(* Usage : 
fbDAIKIN_MasterStation_III_No_1 : FB_BACnet_DAIKIN_MasterStation_III_No_1 :=(Client:=(nDeviceInstance := 1)); 
*)
FUNCTION_BLOCK  FB_BACnet_DAIKIN_MasterStation_III_No_1
VAR_INPUT CONSTANT
	Client : FB_BACnet_Client := (tReadCycleTime:=T#10S,nMaxParallelRequests:=20);
	DAIKIN_MasterStation_III_No_1: FB_BACnetRM_Device := (Client:=Client);
	StartStopCommand_000: FB_BACnetRM_BO := (Client:=Client,nObjectInstance:=1);
	StartStopStatus_000: FB_BACnetRM_BI := (Client:=Client,nObjectInstance:=2);
	Alarm_000: FB_BACnetRM_BI := (Client:=Client,nObjectInstance:=3);
	MalfunctionCode_000: FB_BACnetRM_MI := (Client:=Client,nObjectInstance:=4);
	
	
	
	
	RoomTemp_000: FB_BACnetRM_AI := (Client:=Client,nObjectInstance:=9);
	TempAdjust_000: FB_BACnetRM_AV := (Client:=Client,nObjectInstance:=10);
	FilterSign_000: FB_BACnetRM_BI := (Client:=Client,nObjectInstance:=11);
	FilterSignReset_000: FB_BACnetRM_BV := (Client:=Client,nObjectInstance:=12);
	RemoteControlStart_000: FB_BACnetRM_BV := (Client:=Client,nObjectInstance:=13);
	
	RemoteControlTempAdjust_000: FB_BACnetRM_BV := (Client:=Client,nObjectInstance:=16);
	
	
	
	
	
	
	
	
	
	
	
	
	StartStopCommand_001: FB_BACnetRM_BO := (Client:=Client,nObjectInstance:=257);
	StartStopStatus_001: FB_BACnetRM_BI := (Client:=Client,nObjectInstance:=258);
	Alarm_001: FB_BACnetRM_BI := (Client:=Client,nObjectInstance:=259);
	MalfunctionCode_001: FB_BACnetRM_MI := (Client:=Client,nObjectInstance:=260);
	
	
	
	
	RoomTemp_001: FB_BACnetRM_AI := (Client:=Client,nObjectInstance:=265);
	TempAdjust_001: FB_BACnetRM_AV := (Client:=Client,nObjectInstance:=266);
	FilterSign_001: FB_BACnetRM_BI := (Client:=Client,nObjectInstance:=267);
	FilterSignReset_001: FB_BACnetRM_BV := (Client:=Client,nObjectInstance:=268);
	RemoteControlStart_001: FB_BACnetRM_BV := (Client:=Client,nObjectInstance:=269);
	
	RemoteControlTempAdjust_001: FB_BACnetRM_BV := (Client:=Client,nObjectInstance:=272);
	
	
	
	
	
	
	
	
	
	
	
	
	StartStopCommand_002: FB_BACnetRM_BO := (Client:=Client,nObjectInstance:=513);
	StartStopStatus_002: FB_BACnetRM_BI := (Client:=Client,nObjectInstance:=514);
	Alarm_002: FB_BACnetRM_BI := (Client:=Client,nObjectInstance:=515);
	MalfunctionCode_002: FB_BACnetRM_MI := (Client:=Client,nObjectInstance:=516);
	
	
	
	
	RoomTemp_002: FB_BACnetRM_AI := (Client:=Client,nObjectInstance:=521);
	TempAdjust_002: FB_BACnetRM_AV := (Client:=Client,nObjectInstance:=522);
	FilterSign_002: FB_BACnetRM_BI := (Client:=Client,nObjectInstance:=523);
	FilterSignReset_002: FB_BACnetRM_BV := (Client:=Client,nObjectInstance:=524);
	RemoteControlStart_002: FB_BACnetRM_BV := (Client:=Client,nObjectInstance:=525);
	
	RemoteControlTempAdjust_002: FB_BACnetRM_BV := (Client:=Client,nObjectInstance:=528);
	
	
	
	
	
	
	
	
	
	
	
	
	StartStopCommand_003: FB_BACnetRM_BO := (Client:=Client,nObjectInstance:=769);
	StartStopStatus_003: FB_BACnetRM_BI := (Client:=Client,nObjectInstance:=770);
	Alarm_003: FB_BACnetRM_BI := (Client:=Client,nObjectInstance:=771);
	MalfunctionCode_003: FB_BACnetRM_MI := (Client:=Client,nObjectInstance:=772);
	
	
	
	
	RoomTemp_003: FB_BACnetRM_AI := (Client:=Client,nObjectInstance:=777);
	TempAdjust_003: FB_BACnetRM_AV := (Client:=Client,nObjectInstance:=778);
	FilterSign_003: FB_BACnetRM_BI := (Client:=Client,nObjectInstance:=779);
	FilterSignReset_003: FB_BACnetRM_BV := (Client:=Client,nObjectInstance:=780);
	RemoteControlStart_003: FB_BACnetRM_BV := (Client:=Client,nObjectInstance:=781);
	
	RemoteControlTempAdjust_003: FB_BACnetRM_BV := (Client:=Client,nObjectInstance:=784);
	
	
	
	
	
	
	
	
	
	
	
	
	StartStopCommand_004: FB_BACnetRM_BO := (Client:=Client,nObjectInstance:=1025);
	StartStopStatus_004: FB_BACnetRM_BI := (Client:=Client,nObjectInstance:=1026);
	Alarm_004: FB_BACnetRM_BI := (Client:=Client,nObjectInstance:=1027);
	MalfunctionCode_004: FB_BACnetRM_MI := (Client:=Client,nObjectInstance:=1028);
	
	
	
	
	RoomTemp_004: FB_BACnetRM_AI := (Client:=Client,nObjectInstance:=1033);
	TempAdjust_004: FB_BACnetRM_AV := (Client:=Client,nObjectInstance:=1034);
	FilterSign_004: FB_BACnetRM_BI := (Client:=Client,nObjectInstance:=1035);
	FilterSignReset_004: FB_BACnetRM_BV := (Client:=Client,nObjectInstance:=1036);
	RemoteControlStart_004: FB_BACnetRM_BV := (Client:=Client,nObjectInstance:=1037);
	
	RemoteControlTempAdjust_004: FB_BACnetRM_BV := (Client:=Client,nObjectInstance:=1040);
	
	
	
	
	
	
	
	
	
	
	
	
	StartStopCommand_005: FB_BACnetRM_BO := (Client:=Client,nObjectInstance:=1281);
	StartStopStatus_005: FB_BACnetRM_BI := (Client:=Client,nObjectInstance:=1282);
	Alarm_005: FB_BACnetRM_BI := (Client:=Client,nObjectInstance:=1283);
	MalfunctionCode_005: FB_BACnetRM_MI := (Client:=Client,nObjectInstance:=1284);
	
	
	
	
	RoomTemp_005: FB_BACnetRM_AI := (Client:=Client,nObjectInstance:=1289);
	TempAdjust_005: FB_BACnetRM_AV := (Client:=Client,nObjectInstance:=1290);
	FilterSign_005: FB_BACnetRM_BI := (Client:=Client,nObjectInstance:=1291);
	FilterSignReset_005: FB_BACnetRM_BV := (Client:=Client,nObjectInstance:=1292);
	RemoteControlStart_005: FB_BACnetRM_BV := (Client:=Client,nObjectInstance:=1293);
	
	RemoteControlTempAdjust_005: FB_BACnetRM_BV := (Client:=Client,nObjectInstance:=1296);
	
	
	
	
	
	
	
	
	
	
	
	
	StartStopCommand_006: FB_BACnetRM_BO := (Client:=Client,nObjectInstance:=1537);
	StartStopStatus_006: FB_BACnetRM_BI := (Client:=Client,nObjectInstance:=1538);
	Alarm_006: FB_BACnetRM_BI := (Client:=Client,nObjectInstance:=1539);
	MalfunctionCode_006: FB_BACnetRM_MI := (Client:=Client,nObjectInstance:=1540);
	
	
	
	
	RoomTemp_006: FB_BACnetRM_AI := (Client:=Client,nObjectInstance:=1545);
	TempAdjust_006: FB_BACnetRM_AV := (Client:=Client,nObjectInstance:=1546);
	FilterSign_006: FB_BACnetRM_BI := (Client:=Client,nObjectInstance:=1547);
	FilterSignReset_006: FB_BACnetRM_BV := (Client:=Client,nObjectInstance:=1548);
	RemoteControlStart_006: FB_BACnetRM_BV := (Client:=Client,nObjectInstance:=1549);
	
	RemoteControlTempAdjust_006: FB_BACnetRM_BV := (Client:=Client,nObjectInstance:=1552);
	
	
	
	
	
	
	
	
	
	
	
	
	StartStopCommand_007: FB_BACnetRM_BO := (Client:=Client,nObjectInstance:=1793);
	StartStopStatus_007: FB_BACnetRM_BI := (Client:=Client,nObjectInstance:=1794);
	Alarm_007: FB_BACnetRM_BI := (Client:=Client,nObjectInstance:=1795);
	MalfunctionCode_007: FB_BACnetRM_MI := (Client:=Client,nObjectInstance:=1796);
	
	
	
	
	RoomTemp_007: FB_BACnetRM_AI := (Client:=Client,nObjectInstance:=1801);
	TempAdjust_007: FB_BACnetRM_AV := (Client:=Client,nObjectInstance:=1802);
	FilterSign_007: FB_BACnetRM_BI := (Client:=Client,nObjectInstance:=1803);
	FilterSignReset_007: FB_BACnetRM_BV := (Client:=Client,nObjectInstance:=1804);
	RemoteControlStart_007: FB_BACnetRM_BV := (Client:=Client,nObjectInstance:=1805);
	
	RemoteControlTempAdjust_007: FB_BACnetRM_BV := (Client:=Client,nObjectInstance:=1808);
	
	
	
	
	
	
	
	
	
	
	
	
	StartStopCommand_008: FB_BACnetRM_BO := (Client:=Client,nObjectInstance:=2049);
	StartStopStatus_008: FB_BACnetRM_BI := (Client:=Client,nObjectInstance:=2050);
	Alarm_008: FB_BACnetRM_BI := (Client:=Client,nObjectInstance:=2051);
	MalfunctionCode_008: FB_BACnetRM_MI := (Client:=Client,nObjectInstance:=2052);
	
	
	
	
	RoomTemp_008: FB_BACnetRM_AI := (Client:=Client,nObjectInstance:=2057);
	TempAdjust_008: FB_BACnetRM_AV := (Client:=Client,nObjectInstance:=2058);
	FilterSign_008: FB_BACnetRM_BI := (Client:=Client,nObjectInstance:=2059);
	FilterSignReset_008: FB_BACnetRM_BV := (Client:=Client,nObjectInstance:=2060);
	RemoteControlStart_008: FB_BACnetRM_BV := (Client:=Client,nObjectInstance:=2061);
	
	RemoteControlTempAdjust_008: FB_BACnetRM_BV := (Client:=Client,nObjectInstance:=2064);
	
	
	
	
	
	
	
	
	
	
	
	
	StartStopCommand_009: FB_BACnetRM_BO := (Client:=Client,nObjectInstance:=2305);
	StartStopStatus_009: FB_BACnetRM_BI := (Client:=Client,nObjectInstance:=2306);
	Alarm_009: FB_BACnetRM_BI := (Client:=Client,nObjectInstance:=2307);
	MalfunctionCode_009: FB_BACnetRM_MI := (Client:=Client,nObjectInstance:=2308);
	
	
	
	
	RoomTemp_009: FB_BACnetRM_AI := (Client:=Client,nObjectInstance:=2313);
	TempAdjust_009: FB_BACnetRM_AV := (Client:=Client,nObjectInstance:=2314);
	FilterSign_009: FB_BACnetRM_BI := (Client:=Client,nObjectInstance:=2315);
	FilterSignReset_009: FB_BACnetRM_BV := (Client:=Client,nObjectInstance:=2316);
	RemoteControlStart_009: FB_BACnetRM_BV := (Client:=Client,nObjectInstance:=2317);
	
	RemoteControlTempAdjust_009: FB_BACnetRM_BV := (Client:=Client,nObjectInstance:=2320);
	
	
	
	
	
	
	
	
	
	
	
	
	StartStopCommand_010: FB_BACnetRM_BO := (Client:=Client,nObjectInstance:=2561);
	StartStopStatus_010: FB_BACnetRM_BI := (Client:=Client,nObjectInstance:=2562);
	Alarm_010: FB_BACnetRM_BI := (Client:=Client,nObjectInstance:=2563);
	MalfunctionCode_010: FB_BACnetRM_MI := (Client:=Client,nObjectInstance:=2564);
	
	
	
	
	RoomTemp_010: FB_BACnetRM_AI := (Client:=Client,nObjectInstance:=2569);
	TempAdjust_010: FB_BACnetRM_AV := (Client:=Client,nObjectInstance:=2570);
	FilterSign_010: FB_BACnetRM_BI := (Client:=Client,nObjectInstance:=2571);
	FilterSignReset_010: FB_BACnetRM_BV := (Client:=Client,nObjectInstance:=2572);
	RemoteControlStart_010: FB_BACnetRM_BV := (Client:=Client,nObjectInstance:=2573);
	
	RemoteControlTempAdjust_010: FB_BACnetRM_BV := (Client:=Client,nObjectInstance:=2576);
	
	
	
	
	
	
	
	
	
	
	
	
	StartStopCommand_011: FB_BACnetRM_BO := (Client:=Client,nObjectInstance:=2817);
	StartStopStatus_011: FB_BACnetRM_BI := (Client:=Client,nObjectInstance:=2818);
	Alarm_011: FB_BACnetRM_BI := (Client:=Client,nObjectInstance:=2819);
	MalfunctionCode_011: FB_BACnetRM_MI := (Client:=Client,nObjectInstance:=2820);
	
	
	
	
	RoomTemp_011: FB_BACnetRM_AI := (Client:=Client,nObjectInstance:=2825);
	TempAdjust_011: FB_BACnetRM_AV := (Client:=Client,nObjectInstance:=2826);
	FilterSign_011: FB_BACnetRM_BI := (Client:=Client,nObjectInstance:=2827);
	FilterSignReset_011: FB_BACnetRM_BV := (Client:=Client,nObjectInstance:=2828);
	RemoteControlStart_011: FB_BACnetRM_BV := (Client:=Client,nObjectInstance:=2829);
	
	RemoteControlTempAdjust_011: FB_BACnetRM_BV := (Client:=Client,nObjectInstance:=2832);
	
	
	
	
	
	
	
	
	
	
	
	
	StartStopCommand_012: FB_BACnetRM_BO := (Client:=Client,nObjectInstance:=3073);
	StartStopStatus_012: FB_BACnetRM_BI := (Client:=Client,nObjectInstance:=3074);
	Alarm_012: FB_BACnetRM_BI := (Client:=Client,nObjectInstance:=3075);
	MalfunctionCode_012: FB_BACnetRM_MI := (Client:=Client,nObjectInstance:=3076);
	
	
	
	
	RoomTemp_012: FB_BACnetRM_AI := (Client:=Client,nObjectInstance:=3081);
	TempAdjust_012: FB_BACnetRM_AV := (Client:=Client,nObjectInstance:=3082);
	FilterSign_012: FB_BACnetRM_BI := (Client:=Client,nObjectInstance:=3083);
	FilterSignReset_012: FB_BACnetRM_BV := (Client:=Client,nObjectInstance:=3084);
	RemoteControlStart_012: FB_BACnetRM_BV := (Client:=Client,nObjectInstance:=3085);
	
	RemoteControlTempAdjust_012: FB_BACnetRM_BV := (Client:=Client,nObjectInstance:=3088);
	
	
	
	
	
	
	
	
	
	
	
	
	StartStopCommand_013: FB_BACnetRM_BO := (Client:=Client,nObjectInstance:=3329);
	StartStopStatus_013: FB_BACnetRM_BI := (Client:=Client,nObjectInstance:=3330);
	Alarm_013: FB_BACnetRM_BI := (Client:=Client,nObjectInstance:=3331);
	MalfunctionCode_013: FB_BACnetRM_MI := (Client:=Client,nObjectInstance:=3332);
	
	
	
	
	RoomTemp_013: FB_BACnetRM_AI := (Client:=Client,nObjectInstance:=3337);
	TempAdjust_013: FB_BACnetRM_AV := (Client:=Client,nObjectInstance:=3338);
	FilterSign_013: FB_BACnetRM_BI := (Client:=Client,nObjectInstance:=3339);
	FilterSignReset_013: FB_BACnetRM_BV := (Client:=Client,nObjectInstance:=3340);
	RemoteControlStart_013: FB_BACnetRM_BV := (Client:=Client,nObjectInstance:=3341);
	
	RemoteControlTempAdjust_013: FB_BACnetRM_BV := (Client:=Client,nObjectInstance:=3344);
	
	
	
	
	
	
	
	
	
	
	
	
	StartStopCommand_014: FB_BACnetRM_BO := (Client:=Client,nObjectInstance:=3585);
	StartStopStatus_014: FB_BACnetRM_BI := (Client:=Client,nObjectInstance:=3586);
	Alarm_014: FB_BACnetRM_BI := (Client:=Client,nObjectInstance:=3587);
	MalfunctionCode_014: FB_BACnetRM_MI := (Client:=Client,nObjectInstance:=3588);
	
	
	
	
	RoomTemp_014: FB_BACnetRM_AI := (Client:=Client,nObjectInstance:=3593);
	TempAdjust_014: FB_BACnetRM_AV := (Client:=Client,nObjectInstance:=3594);
	FilterSign_014: FB_BACnetRM_BI := (Client:=Client,nObjectInstance:=3595);
	FilterSignReset_014: FB_BACnetRM_BV := (Client:=Client,nObjectInstance:=3596);
	RemoteControlStart_014: FB_BACnetRM_BV := (Client:=Client,nObjectInstance:=3597);
	
	RemoteControlTempAdjust_014: FB_BACnetRM_BV := (Client:=Client,nObjectInstance:=3600);
	
	
	
	
	
	
	
	
	
	
	
	
	StartStopCommand_015: FB_BACnetRM_BO := (Client:=Client,nObjectInstance:=3841);
	StartStopStatus_015: FB_BACnetRM_BI := (Client:=Client,nObjectInstance:=3842);
	Alarm_015: FB_BACnetRM_BI := (Client:=Client,nObjectInstance:=3843);
	MalfunctionCode_015: FB_BACnetRM_MI := (Client:=Client,nObjectInstance:=3844);
	
	
	
	
	RoomTemp_015: FB_BACnetRM_AI := (Client:=Client,nObjectInstance:=3849);
	TempAdjust_015: FB_BACnetRM_AV := (Client:=Client,nObjectInstance:=3850);
	FilterSign_015: FB_BACnetRM_BI := (Client:=Client,nObjectInstance:=3851);
	FilterSignReset_015: FB_BACnetRM_BV := (Client:=Client,nObjectInstance:=3852);
	RemoteControlStart_015: FB_BACnetRM_BV := (Client:=Client,nObjectInstance:=3853);
	
	RemoteControlTempAdjust_015: FB_BACnetRM_BV := (Client:=Client,nObjectInstance:=3856);
	
	
	
	
	
	
	
	
	
	
	
	
	StartStopCommand_016: FB_BACnetRM_BO := (Client:=Client,nObjectInstance:=4097);
	StartStopStatus_016: FB_BACnetRM_BI := (Client:=Client,nObjectInstance:=4098);
	Alarm_016: FB_BACnetRM_BI := (Client:=Client,nObjectInstance:=4099);
	MalfunctionCode_016: FB_BACnetRM_MI := (Client:=Client,nObjectInstance:=4100);
	
	
	
	
	RoomTemp_016: FB_BACnetRM_AI := (Client:=Client,nObjectInstance:=4105);
	TempAdjust_016: FB_BACnetRM_AV := (Client:=Client,nObjectInstance:=4106);
	FilterSign_016: FB_BACnetRM_BI := (Client:=Client,nObjectInstance:=4107);
	FilterSignReset_016: FB_BACnetRM_BV := (Client:=Client,nObjectInstance:=4108);
	RemoteControlStart_016: FB_BACnetRM_BV := (Client:=Client,nObjectInstance:=4109);
	
	RemoteControlTempAdjust_016: FB_BACnetRM_BV := (Client:=Client,nObjectInstance:=4112);
	
	
	
	
	
	
	
	
	
	
	
	
	StartStopCommand_017: FB_BACnetRM_BO := (Client:=Client,nObjectInstance:=4353);
	StartStopStatus_017: FB_BACnetRM_BI := (Client:=Client,nObjectInstance:=4354);
	Alarm_017: FB_BACnetRM_BI := (Client:=Client,nObjectInstance:=4355);
	MalfunctionCode_017: FB_BACnetRM_MI := (Client:=Client,nObjectInstance:=4356);
	
	
	
	
	RoomTemp_017: FB_BACnetRM_AI := (Client:=Client,nObjectInstance:=4361);
	TempAdjust_017: FB_BACnetRM_AV := (Client:=Client,nObjectInstance:=4362);
	FilterSign_017: FB_BACnetRM_BI := (Client:=Client,nObjectInstance:=4363);
	FilterSignReset_017: FB_BACnetRM_BV := (Client:=Client,nObjectInstance:=4364);
	RemoteControlStart_017: FB_BACnetRM_BV := (Client:=Client,nObjectInstance:=4365);
	
	RemoteControlTempAdjust_017: FB_BACnetRM_BV := (Client:=Client,nObjectInstance:=4368);
	
	
	
	
	
	
	
	
	
	
	
	
	StartStopCommand_018: FB_BACnetRM_BO := (Client:=Client,nObjectInstance:=4609);
	StartStopStatus_018: FB_BACnetRM_BI := (Client:=Client,nObjectInstance:=4610);
	Alarm_018: FB_BACnetRM_BI := (Client:=Client,nObjectInstance:=4611);
	MalfunctionCode_018: FB_BACnetRM_MI := (Client:=Client,nObjectInstance:=4612);
	
	
	
	
	RoomTemp_018: FB_BACnetRM_AI := (Client:=Client,nObjectInstance:=4617);
	TempAdjust_018: FB_BACnetRM_AV := (Client:=Client,nObjectInstance:=4618);
	FilterSign_018: FB_BACnetRM_BI := (Client:=Client,nObjectInstance:=4619);
	FilterSignReset_018: FB_BACnetRM_BV := (Client:=Client,nObjectInstance:=4620);
	RemoteControlStart_018: FB_BACnetRM_BV := (Client:=Client,nObjectInstance:=4621);
	
	RemoteControlTempAdjust_018: FB_BACnetRM_BV := (Client:=Client,nObjectInstance:=4624);
	
	
	
	
	
	
	
	
	
	
	
	
	StartStopCommand_019: FB_BACnetRM_BO := (Client:=Client,nObjectInstance:=4865);
	StartStopStatus_019: FB_BACnetRM_BI := (Client:=Client,nObjectInstance:=4866);
	Alarm_019: FB_BACnetRM_BI := (Client:=Client,nObjectInstance:=4867);
	MalfunctionCode_019: FB_BACnetRM_MI := (Client:=Client,nObjectInstance:=4868);
	
	
	
	
	RoomTemp_019: FB_BACnetRM_AI := (Client:=Client,nObjectInstance:=4873);
	TempAdjust_019: FB_BACnetRM_AV := (Client:=Client,nObjectInstance:=4874);
	FilterSign_019: FB_BACnetRM_BI := (Client:=Client,nObjectInstance:=4875);
	FilterSignReset_019: FB_BACnetRM_BV := (Client:=Client,nObjectInstance:=4876);
	RemoteControlStart_019: FB_BACnetRM_BV := (Client:=Client,nObjectInstance:=4877);
	
	RemoteControlTempAdjust_019: FB_BACnetRM_BV := (Client:=Client,nObjectInstance:=4880);
	
	
	
	
	
	
	
	
	
	
	
	
	StartStopCommand_020: FB_BACnetRM_BO := (Client:=Client,nObjectInstance:=5121);
	StartStopStatus_020: FB_BACnetRM_BI := (Client:=Client,nObjectInstance:=5122);
	Alarm_020: FB_BACnetRM_BI := (Client:=Client,nObjectInstance:=5123);
	MalfunctionCode_020: FB_BACnetRM_MI := (Client:=Client,nObjectInstance:=5124);
	
	
	
	
	RoomTemp_020: FB_BACnetRM_AI := (Client:=Client,nObjectInstance:=5129);
	TempAdjust_020: FB_BACnetRM_AV := (Client:=Client,nObjectInstance:=5130);
	FilterSign_020: FB_BACnetRM_BI := (Client:=Client,nObjectInstance:=5131);
	FilterSignReset_020: FB_BACnetRM_BV := (Client:=Client,nObjectInstance:=5132);
	RemoteControlStart_020: FB_BACnetRM_BV := (Client:=Client,nObjectInstance:=5133);
	
	RemoteControlTempAdjust_020: FB_BACnetRM_BV := (Client:=Client,nObjectInstance:=5136);
	
	
	
	
	
	
	
	
	
	
	
	
	StartStopCommand_021: FB_BACnetRM_BO := (Client:=Client,nObjectInstance:=5377);
	StartStopStatus_021: FB_BACnetRM_BI := (Client:=Client,nObjectInstance:=5378);
	Alarm_021: FB_BACnetRM_BI := (Client:=Client,nObjectInstance:=5379);
	MalfunctionCode_021: FB_BACnetRM_MI := (Client:=Client,nObjectInstance:=5380);
	
	
	
	
	RoomTemp_021: FB_BACnetRM_AI := (Client:=Client,nObjectInstance:=5385);
	TempAdjust_021: FB_BACnetRM_AV := (Client:=Client,nObjectInstance:=5386);
	FilterSign_021: FB_BACnetRM_BI := (Client:=Client,nObjectInstance:=5387);
	FilterSignReset_021: FB_BACnetRM_BV := (Client:=Client,nObjectInstance:=5388);
	RemoteControlStart_021: FB_BACnetRM_BV := (Client:=Client,nObjectInstance:=5389);
	
	RemoteControlTempAdjust_021: FB_BACnetRM_BV := (Client:=Client,nObjectInstance:=5392);
	
	
	
	
	
	
	
	
	
	
	
	
	StartStopCommand_022: FB_BACnetRM_BO := (Client:=Client,nObjectInstance:=5633);
	StartStopStatus_022: FB_BACnetRM_BI := (Client:=Client,nObjectInstance:=5634);
	Alarm_022: FB_BACnetRM_BI := (Client:=Client,nObjectInstance:=5635);
	MalfunctionCode_022: FB_BACnetRM_MI := (Client:=Client,nObjectInstance:=5636);
	
	
	
	
	RoomTemp_022: FB_BACnetRM_AI := (Client:=Client,nObjectInstance:=5641);
	TempAdjust_022: FB_BACnetRM_AV := (Client:=Client,nObjectInstance:=5642);
	FilterSign_022: FB_BACnetRM_BI := (Client:=Client,nObjectInstance:=5643);
	FilterSignReset_022: FB_BACnetRM_BV := (Client:=Client,nObjectInstance:=5644);
	RemoteControlStart_022: FB_BACnetRM_BV := (Client:=Client,nObjectInstance:=5645);
	
	RemoteControlTempAdjust_022: FB_BACnetRM_BV := (Client:=Client,nObjectInstance:=5648);
	
	
	
	
	
	
	
	
	
	
	
	
	StartStopCommand_023: FB_BACnetRM_BO := (Client:=Client,nObjectInstance:=5889);
	StartStopStatus_023: FB_BACnetRM_BI := (Client:=Client,nObjectInstance:=5890);
	Alarm_023: FB_BACnetRM_BI := (Client:=Client,nObjectInstance:=5891);
	MalfunctionCode_023: FB_BACnetRM_MI := (Client:=Client,nObjectInstance:=5892);
	
	
	
	
	RoomTemp_023: FB_BACnetRM_AI := (Client:=Client,nObjectInstance:=5897);
	TempAdjust_023: FB_BACnetRM_AV := (Client:=Client,nObjectInstance:=5898);
	FilterSign_023: FB_BACnetRM_BI := (Client:=Client,nObjectInstance:=5899);
	FilterSignReset_023: FB_BACnetRM_BV := (Client:=Client,nObjectInstance:=5900);
	RemoteControlStart_023: FB_BACnetRM_BV := (Client:=Client,nObjectInstance:=5901);
	
	RemoteControlTempAdjust_023: FB_BACnetRM_BV := (Client:=Client,nObjectInstance:=5904);
	
	
	
	
	
	
	
	
	
	
	
	
	StartStopCommand_024: FB_BACnetRM_BO := (Client:=Client,nObjectInstance:=6145);
	StartStopStatus_024: FB_BACnetRM_BI := (Client:=Client,nObjectInstance:=6146);
	Alarm_024: FB_BACnetRM_BI := (Client:=Client,nObjectInstance:=6147);
	MalfunctionCode_024: FB_BACnetRM_MI := (Client:=Client,nObjectInstance:=6148);
	
	
	
	
	RoomTemp_024: FB_BACnetRM_AI := (Client:=Client,nObjectInstance:=6153);
	TempAdjust_024: FB_BACnetRM_AV := (Client:=Client,nObjectInstance:=6154);
	FilterSign_024: FB_BACnetRM_BI := (Client:=Client,nObjectInstance:=6155);
	FilterSignReset_024: FB_BACnetRM_BV := (Client:=Client,nObjectInstance:=6156);
	RemoteControlStart_024: FB_BACnetRM_BV := (Client:=Client,nObjectInstance:=6157);
	
	RemoteControlTempAdjust_024: FB_BACnetRM_BV := (Client:=Client,nObjectInstance:=6160);
	
	
	
	
	
	
	
	
	
	
	
	
	StartStopCommand_025: FB_BACnetRM_BO := (Client:=Client,nObjectInstance:=6401);
	StartStopStatus_025: FB_BACnetRM_BI := (Client:=Client,nObjectInstance:=6402);
	Alarm_025: FB_BACnetRM_BI := (Client:=Client,nObjectInstance:=6403);
	MalfunctionCode_025: FB_BACnetRM_MI := (Client:=Client,nObjectInstance:=6404);
	
	
	
	
	RoomTemp_025: FB_BACnetRM_AI := (Client:=Client,nObjectInstance:=6409);
	TempAdjust_025: FB_BACnetRM_AV := (Client:=Client,nObjectInstance:=6410);
	FilterSign_025: FB_BACnetRM_BI := (Client:=Client,nObjectInstance:=6411);
	FilterSignReset_025: FB_BACnetRM_BV := (Client:=Client,nObjectInstance:=6412);
	RemoteControlStart_025: FB_BACnetRM_BV := (Client:=Client,nObjectInstance:=6413);
	
	RemoteControlTempAdjust_025: FB_BACnetRM_BV := (Client:=Client,nObjectInstance:=6416);
	
	
	
	
	
	
	
	
	
	
	
	
	StartStopCommand_026: FB_BACnetRM_BO := (Client:=Client,nObjectInstance:=6657);
	StartStopStatus_026: FB_BACnetRM_BI := (Client:=Client,nObjectInstance:=6658);
	Alarm_026: FB_BACnetRM_BI := (Client:=Client,nObjectInstance:=6659);
	MalfunctionCode_026: FB_BACnetRM_MI := (Client:=Client,nObjectInstance:=6660);
	
	
	
	
	RoomTemp_026: FB_BACnetRM_AI := (Client:=Client,nObjectInstance:=6665);
	TempAdjust_026: FB_BACnetRM_AV := (Client:=Client,nObjectInstance:=6666);
	FilterSign_026: FB_BACnetRM_BI := (Client:=Client,nObjectInstance:=6667);
	FilterSignReset_026: FB_BACnetRM_BV := (Client:=Client,nObjectInstance:=6668);
	RemoteControlStart_026: FB_BACnetRM_BV := (Client:=Client,nObjectInstance:=6669);
	
	RemoteControlTempAdjust_026: FB_BACnetRM_BV := (Client:=Client,nObjectInstance:=6672);
	
	
	
	
	
	
	
	
	
	
	
	
	StartStopCommand_027: FB_BACnetRM_BO := (Client:=Client,nObjectInstance:=6913);
	StartStopStatus_027: FB_BACnetRM_BI := (Client:=Client,nObjectInstance:=6914);
	Alarm_027: FB_BACnetRM_BI := (Client:=Client,nObjectInstance:=6915);
	MalfunctionCode_027: FB_BACnetRM_MI := (Client:=Client,nObjectInstance:=6916);
	
	
	
	
	RoomTemp_027: FB_BACnetRM_AI := (Client:=Client,nObjectInstance:=6921);
	TempAdjust_027: FB_BACnetRM_AV := (Client:=Client,nObjectInstance:=6922);
	FilterSign_027: FB_BACnetRM_BI := (Client:=Client,nObjectInstance:=6923);
	FilterSignReset_027: FB_BACnetRM_BV := (Client:=Client,nObjectInstance:=6924);
	RemoteControlStart_027: FB_BACnetRM_BV := (Client:=Client,nObjectInstance:=6925);
	
	RemoteControlTempAdjust_027: FB_BACnetRM_BV := (Client:=Client,nObjectInstance:=6928);
	
	
	
	
	
	
	
	
	
	
	
	
	StartStopCommand_028: FB_BACnetRM_BO := (Client:=Client,nObjectInstance:=7169);
	StartStopStatus_028: FB_BACnetRM_BI := (Client:=Client,nObjectInstance:=7170);
	Alarm_028: FB_BACnetRM_BI := (Client:=Client,nObjectInstance:=7171);
	MalfunctionCode_028: FB_BACnetRM_MI := (Client:=Client,nObjectInstance:=7172);
	
	
	
	
	RoomTemp_028: FB_BACnetRM_AI := (Client:=Client,nObjectInstance:=7177);
	TempAdjust_028: FB_BACnetRM_AV := (Client:=Client,nObjectInstance:=7178);
	FilterSign_028: FB_BACnetRM_BI := (Client:=Client,nObjectInstance:=7179);
	FilterSignReset_028: FB_BACnetRM_BV := (Client:=Client,nObjectInstance:=7180);
	RemoteControlStart_028: FB_BACnetRM_BV := (Client:=Client,nObjectInstance:=7181);
	
	RemoteControlTempAdjust_028: FB_BACnetRM_BV := (Client:=Client,nObjectInstance:=7184);
	
	
	
	
	
	
	
	
	
	
	
	
	StartStopCommand_029: FB_BACnetRM_BO := (Client:=Client,nObjectInstance:=7425);
	StartStopStatus_029: FB_BACnetRM_BI := (Client:=Client,nObjectInstance:=7426);
	Alarm_029: FB_BACnetRM_BI := (Client:=Client,nObjectInstance:=7427);
	MalfunctionCode_029: FB_BACnetRM_MI := (Client:=Client,nObjectInstance:=7428);
	
	
	
	
	RoomTemp_029: FB_BACnetRM_AI := (Client:=Client,nObjectInstance:=7433);
	TempAdjust_029: FB_BACnetRM_AV := (Client:=Client,nObjectInstance:=7434);
	FilterSign_029: FB_BACnetRM_BI := (Client:=Client,nObjectInstance:=7435);
	FilterSignReset_029: FB_BACnetRM_BV := (Client:=Client,nObjectInstance:=7436);
	RemoteControlStart_029: FB_BACnetRM_BV := (Client:=Client,nObjectInstance:=7437);
	
	RemoteControlTempAdjust_029: FB_BACnetRM_BV := (Client:=Client,nObjectInstance:=7440);
	
	
	
	
	
	
	
	
	
	
	
	
	StartStopCommand_030: FB_BACnetRM_BO := (Client:=Client,nObjectInstance:=7681);
	StartStopStatus_030: FB_BACnetRM_BI := (Client:=Client,nObjectInstance:=7682);
	Alarm_030: FB_BACnetRM_BI := (Client:=Client,nObjectInstance:=7683);
	MalfunctionCode_030: FB_BACnetRM_MI := (Client:=Client,nObjectInstance:=7684);
	
	
	
	
	RoomTemp_030: FB_BACnetRM_AI := (Client:=Client,nObjectInstance:=7689);
	TempAdjust_030: FB_BACnetRM_AV := (Client:=Client,nObjectInstance:=7690);
	FilterSign_030: FB_BACnetRM_BI := (Client:=Client,nObjectInstance:=7691);
	FilterSignReset_030: FB_BACnetRM_BV := (Client:=Client,nObjectInstance:=7692);
	RemoteControlStart_030: FB_BACnetRM_BV := (Client:=Client,nObjectInstance:=7693);
	
	RemoteControlTempAdjust_030: FB_BACnetRM_BV := (Client:=Client,nObjectInstance:=7696);
	
	
	
	
	
	
	
	
	
	
	
	
	StartStopCommand_031: FB_BACnetRM_BO := (Client:=Client,nObjectInstance:=7937);
	StartStopStatus_031: FB_BACnetRM_BI := (Client:=Client,nObjectInstance:=7938);
	Alarm_031: FB_BACnetRM_BI := (Client:=Client,nObjectInstance:=7939);
	MalfunctionCode_031: FB_BACnetRM_MI := (Client:=Client,nObjectInstance:=7940);
	
	
	
	
	RoomTemp_031: FB_BACnetRM_AI := (Client:=Client,nObjectInstance:=7945);
	TempAdjust_031: FB_BACnetRM_AV := (Client:=Client,nObjectInstance:=7946);
	FilterSign_031: FB_BACnetRM_BI := (Client:=Client,nObjectInstance:=7947);
	FilterSignReset_031: FB_BACnetRM_BV := (Client:=Client,nObjectInstance:=7948);
	RemoteControlStart_031: FB_BACnetRM_BV := (Client:=Client,nObjectInstance:=7949);
	
	RemoteControlTempAdjust_031: FB_BACnetRM_BV := (Client:=Client,nObjectInstance:=7952);
	
	
	
	
	
	
	
	
	
	
	
	
	StartStopCommand_032: FB_BACnetRM_BO := (Client:=Client,nObjectInstance:=8193);
	StartStopStatus_032: FB_BACnetRM_BI := (Client:=Client,nObjectInstance:=8194);
	Alarm_032: FB_BACnetRM_BI := (Client:=Client,nObjectInstance:=8195);
	MalfunctionCode_032: FB_BACnetRM_MI := (Client:=Client,nObjectInstance:=8196);
	
	
	
	
	RoomTemp_032: FB_BACnetRM_AI := (Client:=Client,nObjectInstance:=8201);
	TempAdjust_032: FB_BACnetRM_AV := (Client:=Client,nObjectInstance:=8202);
	FilterSign_032: FB_BACnetRM_BI := (Client:=Client,nObjectInstance:=8203);
	FilterSignReset_032: FB_BACnetRM_BV := (Client:=Client,nObjectInstance:=8204);
	RemoteControlStart_032: FB_BACnetRM_BV := (Client:=Client,nObjectInstance:=8205);
	
	RemoteControlTempAdjust_032: FB_BACnetRM_BV := (Client:=Client,nObjectInstance:=8208);
	
	
	
	
	
	
	
	
	
	
	
	
	StartStopCommand_033: FB_BACnetRM_BO := (Client:=Client,nObjectInstance:=8449);
	StartStopStatus_033: FB_BACnetRM_BI := (Client:=Client,nObjectInstance:=8450);
	Alarm_033: FB_BACnetRM_BI := (Client:=Client,nObjectInstance:=8451);
	MalfunctionCode_033: FB_BACnetRM_MI := (Client:=Client,nObjectInstance:=8452);
	
	
	
	
	RoomTemp_033: FB_BACnetRM_AI := (Client:=Client,nObjectInstance:=8457);
	TempAdjust_033: FB_BACnetRM_AV := (Client:=Client,nObjectInstance:=8458);
	FilterSign_033: FB_BACnetRM_BI := (Client:=Client,nObjectInstance:=8459);
	FilterSignReset_033: FB_BACnetRM_BV := (Client:=Client,nObjectInstance:=8460);
	RemoteControlStart_033: FB_BACnetRM_BV := (Client:=Client,nObjectInstance:=8461);
	
	RemoteControlTempAdjust_033: FB_BACnetRM_BV := (Client:=Client,nObjectInstance:=8464);
	
	
	
	
	
	
	
	
	
	
	
	
	StartStopCommand_034: FB_BACnetRM_BO := (Client:=Client,nObjectInstance:=8705);
	StartStopStatus_034: FB_BACnetRM_BI := (Client:=Client,nObjectInstance:=8706);
	Alarm_034: FB_BACnetRM_BI := (Client:=Client,nObjectInstance:=8707);
	MalfunctionCode_034: FB_BACnetRM_MI := (Client:=Client,nObjectInstance:=8708);
	
	
	
	
	RoomTemp_034: FB_BACnetRM_AI := (Client:=Client,nObjectInstance:=8713);
	TempAdjust_034: FB_BACnetRM_AV := (Client:=Client,nObjectInstance:=8714);
	FilterSign_034: FB_BACnetRM_BI := (Client:=Client,nObjectInstance:=8715);
	FilterSignReset_034: FB_BACnetRM_BV := (Client:=Client,nObjectInstance:=8716);
	RemoteControlStart_034: FB_BACnetRM_BV := (Client:=Client,nObjectInstance:=8717);
	
	RemoteControlTempAdjust_034: FB_BACnetRM_BV := (Client:=Client,nObjectInstance:=8720);
	
	
	
	
	
	
	
	
	
	
	
	
	StartStopCommand_035: FB_BACnetRM_BO := (Client:=Client,nObjectInstance:=8961);
	StartStopStatus_035: FB_BACnetRM_BI := (Client:=Client,nObjectInstance:=8962);
	Alarm_035: FB_BACnetRM_BI := (Client:=Client,nObjectInstance:=8963);
	MalfunctionCode_035: FB_BACnetRM_MI := (Client:=Client,nObjectInstance:=8964);
	
	
	
	
	RoomTemp_035: FB_BACnetRM_AI := (Client:=Client,nObjectInstance:=8969);
	TempAdjust_035: FB_BACnetRM_AV := (Client:=Client,nObjectInstance:=8970);
	FilterSign_035: FB_BACnetRM_BI := (Client:=Client,nObjectInstance:=8971);
	FilterSignReset_035: FB_BACnetRM_BV := (Client:=Client,nObjectInstance:=8972);
	RemoteControlStart_035: FB_BACnetRM_BV := (Client:=Client,nObjectInstance:=8973);
	
	RemoteControlTempAdjust_035: FB_BACnetRM_BV := (Client:=Client,nObjectInstance:=8976);
	
	
	
	
	
	
	
	
	
	
	
	
	StartStopCommand_036: FB_BACnetRM_BO := (Client:=Client,nObjectInstance:=9217);
	StartStopStatus_036: FB_BACnetRM_BI := (Client:=Client,nObjectInstance:=9218);
	Alarm_036: FB_BACnetRM_BI := (Client:=Client,nObjectInstance:=9219);
	MalfunctionCode_036: FB_BACnetRM_MI := (Client:=Client,nObjectInstance:=9220);
	
	
	
	
	RoomTemp_036: FB_BACnetRM_AI := (Client:=Client,nObjectInstance:=9225);
	TempAdjust_036: FB_BACnetRM_AV := (Client:=Client,nObjectInstance:=9226);
	FilterSign_036: FB_BACnetRM_BI := (Client:=Client,nObjectInstance:=9227);
	FilterSignReset_036: FB_BACnetRM_BV := (Client:=Client,nObjectInstance:=9228);
	RemoteControlStart_036: FB_BACnetRM_BV := (Client:=Client,nObjectInstance:=9229);
	
	RemoteControlTempAdjust_036: FB_BACnetRM_BV := (Client:=Client,nObjectInstance:=9232);
	
	
	
	
	
	
	
	
	
	
	
	
	StartStopCommand_037: FB_BACnetRM_BO := (Client:=Client,nObjectInstance:=9473);
	StartStopStatus_037: FB_BACnetRM_BI := (Client:=Client,nObjectInstance:=9474);
	Alarm_037: FB_BACnetRM_BI := (Client:=Client,nObjectInstance:=9475);
	MalfunctionCode_037: FB_BACnetRM_MI := (Client:=Client,nObjectInstance:=9476);
	
	
	
	
	RoomTemp_037: FB_BACnetRM_AI := (Client:=Client,nObjectInstance:=9481);
	TempAdjust_037: FB_BACnetRM_AV := (Client:=Client,nObjectInstance:=9482);
	FilterSign_037: FB_BACnetRM_BI := (Client:=Client,nObjectInstance:=9483);
	FilterSignReset_037: FB_BACnetRM_BV := (Client:=Client,nObjectInstance:=9484);
	RemoteControlStart_037: FB_BACnetRM_BV := (Client:=Client,nObjectInstance:=9485);
	
	RemoteControlTempAdjust_037: FB_BACnetRM_BV := (Client:=Client,nObjectInstance:=9488);
	
	
	
	
	
	
	
	
	
	
	
	
	StartStopCommand_038: FB_BACnetRM_BO := (Client:=Client,nObjectInstance:=9729);
	StartStopStatus_038: FB_BACnetRM_BI := (Client:=Client,nObjectInstance:=9730);
	Alarm_038: FB_BACnetRM_BI := (Client:=Client,nObjectInstance:=9731);
	MalfunctionCode_038: FB_BACnetRM_MI := (Client:=Client,nObjectInstance:=9732);
	
	
	
	
	RoomTemp_038: FB_BACnetRM_AI := (Client:=Client,nObjectInstance:=9737);
	TempAdjust_038: FB_BACnetRM_AV := (Client:=Client,nObjectInstance:=9738);
	FilterSign_038: FB_BACnetRM_BI := (Client:=Client,nObjectInstance:=9739);
	FilterSignReset_038: FB_BACnetRM_BV := (Client:=Client,nObjectInstance:=9740);
	RemoteControlStart_038: FB_BACnetRM_BV := (Client:=Client,nObjectInstance:=9741);
	
	RemoteControlTempAdjust_038: FB_BACnetRM_BV := (Client:=Client,nObjectInstance:=9744);
	
	
	
	
	
	
	
	
	
	
	
	
	StartStopCommand_039: FB_BACnetRM_BO := (Client:=Client,nObjectInstance:=9985);
	StartStopStatus_039: FB_BACnetRM_BI := (Client:=Client,nObjectInstance:=9986);
	Alarm_039: FB_BACnetRM_BI := (Client:=Client,nObjectInstance:=9987);
	MalfunctionCode_039: FB_BACnetRM_MI := (Client:=Client,nObjectInstance:=9988);
	
	
	
	
	RoomTemp_039: FB_BACnetRM_AI := (Client:=Client,nObjectInstance:=9993);
	TempAdjust_039: FB_BACnetRM_AV := (Client:=Client,nObjectInstance:=9994);
	FilterSign_039: FB_BACnetRM_BI := (Client:=Client,nObjectInstance:=9995);
	FilterSignReset_039: FB_BACnetRM_BV := (Client:=Client,nObjectInstance:=9996);
	RemoteControlStart_039: FB_BACnetRM_BV := (Client:=Client,nObjectInstance:=9997);
	
	RemoteControlTempAdjust_039: FB_BACnetRM_BV := (Client:=Client,nObjectInstance:=10000);
	
	
	
	
	
	
	
	
	
	
	
	
	StartStopCommand_041: FB_BACnetRM_BO := (Client:=Client,nObjectInstance:=10497);
	StartStopStatus_041: FB_BACnetRM_BI := (Client:=Client,nObjectInstance:=10498);
	Alarm_041: FB_BACnetRM_BI := (Client:=Client,nObjectInstance:=10499);
	MalfunctionCode_041: FB_BACnetRM_MI := (Client:=Client,nObjectInstance:=10500);
	
	
	
	
	RoomTemp_041: FB_BACnetRM_AI := (Client:=Client,nObjectInstance:=10505);
	TempAdjust_041: FB_BACnetRM_AV := (Client:=Client,nObjectInstance:=10506);
	FilterSign_041: FB_BACnetRM_BI := (Client:=Client,nObjectInstance:=10507);
	FilterSignReset_041: FB_BACnetRM_BV := (Client:=Client,nObjectInstance:=10508);
	RemoteControlStart_041: FB_BACnetRM_BV := (Client:=Client,nObjectInstance:=10509);
	
	RemoteControlTempAdjust_041: FB_BACnetRM_BV := (Client:=Client,nObjectInstance:=10512);
	
	
	
	
	
	
	
	
	
	
	
	
	StartStopCommand_042: FB_BACnetRM_BO := (Client:=Client,nObjectInstance:=10753);
	StartStopStatus_042: FB_BACnetRM_BI := (Client:=Client,nObjectInstance:=10754);
	Alarm_042: FB_BACnetRM_BI := (Client:=Client,nObjectInstance:=10755);
	MalfunctionCode_042: FB_BACnetRM_MI := (Client:=Client,nObjectInstance:=10756);
	
	
	
	
	RoomTemp_042: FB_BACnetRM_AI := (Client:=Client,nObjectInstance:=10761);
	TempAdjust_042: FB_BACnetRM_AV := (Client:=Client,nObjectInstance:=10762);
	FilterSign_042: FB_BACnetRM_BI := (Client:=Client,nObjectInstance:=10763);
	FilterSignReset_042: FB_BACnetRM_BV := (Client:=Client,nObjectInstance:=10764);
	RemoteControlStart_042: FB_BACnetRM_BV := (Client:=Client,nObjectInstance:=10765);
	
	RemoteControlTempAdjust_042: FB_BACnetRM_BV := (Client:=Client,nObjectInstance:=10768);
	
	
	
	
	
	
	
	
	
	
	
	
	StartStopCommand_043: FB_BACnetRM_BO := (Client:=Client,nObjectInstance:=11009);
	StartStopStatus_043: FB_BACnetRM_BI := (Client:=Client,nObjectInstance:=11010);
	Alarm_043: FB_BACnetRM_BI := (Client:=Client,nObjectInstance:=11011);
	MalfunctionCode_043: FB_BACnetRM_MI := (Client:=Client,nObjectInstance:=11012);
	
	
	
	
	RoomTemp_043: FB_BACnetRM_AI := (Client:=Client,nObjectInstance:=11017);
	TempAdjust_043: FB_BACnetRM_AV := (Client:=Client,nObjectInstance:=11018);
	FilterSign_043: FB_BACnetRM_BI := (Client:=Client,nObjectInstance:=11019);
	FilterSignReset_043: FB_BACnetRM_BV := (Client:=Client,nObjectInstance:=11020);
	RemoteControlStart_043: FB_BACnetRM_BV := (Client:=Client,nObjectInstance:=11021);
	
	RemoteControlTempAdjust_043: FB_BACnetRM_BV := (Client:=Client,nObjectInstance:=11024);
	
	
	
	
	
	
	
	
	
	
	
	
	//StartStopCommand_044: FB_BACnetRM_BO := (Client:=Client,nObjectInstance:=11265);
	//StartStopStatus_044: FB_BACnetRM_BI := (Client:=Client,nObjectInstance:=11266);
	//Alarm_044: FB_BACnetRM_BI := (Client:=Client,nObjectInstance:=11267);
	//MalfunctionCode_044: FB_BACnetRM_MI := (Client:=Client,nObjectInstance:=11268);
	
	
	
	
	//RoomTemp_044: FB_BACnetRM_AI := (Client:=Client,nObjectInstance:=11273);
	//TempAdjust_044: FB_BACnetRM_AV := (Client:=Client,nObjectInstance:=11274);
	//FilterSign_044: FB_BACnetRM_BI := (Client:=Client,nObjectInstance:=11275);
	//FilterSignReset_044: FB_BACnetRM_BV := (Client:=Client,nObjectInstance:=11276);
	//RemoteControlStart_044: FB_BACnetRM_BV := (Client:=Client,nObjectInstance:=11277);
	//
	//RemoteControlTempAdjust_044: FB_BACnetRM_BV := (Client:=Client,nObjectInstance:=11280);
	
	//
	
	
	
	
	
	
	
	
	
	
	StartStopCommand_045: FB_BACnetRM_BO := (Client:=Client,nObjectInstance:=11521);
	StartStopStatus_045: FB_BACnetRM_BI := (Client:=Client,nObjectInstance:=11522);
	Alarm_045: FB_BACnetRM_BI := (Client:=Client,nObjectInstance:=11523);
	MalfunctionCode_045: FB_BACnetRM_MI := (Client:=Client,nObjectInstance:=11524);
	
	
	
	
	RoomTemp_045: FB_BACnetRM_AI := (Client:=Client,nObjectInstance:=11529);
	TempAdjust_045: FB_BACnetRM_AV := (Client:=Client,nObjectInstance:=11530);
	FilterSign_045: FB_BACnetRM_BI := (Client:=Client,nObjectInstance:=11531);
	FilterSignReset_045: FB_BACnetRM_BV := (Client:=Client,nObjectInstance:=11532);
	RemoteControlStart_045: FB_BACnetRM_BV := (Client:=Client,nObjectInstance:=11533);
	
	RemoteControlTempAdjust_045: FB_BACnetRM_BV := (Client:=Client,nObjectInstance:=11536);
	
	
	
	
	
	
	
	
	
	
	
	
	StartStopCommand_046: FB_BACnetRM_BO := (Client:=Client,nObjectInstance:=11777);
	StartStopStatus_046: FB_BACnetRM_BI := (Client:=Client,nObjectInstance:=11778);
	Alarm_046: FB_BACnetRM_BI := (Client:=Client,nObjectInstance:=11779);
	MalfunctionCode_046: FB_BACnetRM_MI := (Client:=Client,nObjectInstance:=11780);
	
	
	
	
	RoomTemp_046: FB_BACnetRM_AI := (Client:=Client,nObjectInstance:=11785);
	TempAdjust_046: FB_BACnetRM_AV := (Client:=Client,nObjectInstance:=11786);
	FilterSign_046: FB_BACnetRM_BI := (Client:=Client,nObjectInstance:=11787);
	FilterSignReset_046: FB_BACnetRM_BV := (Client:=Client,nObjectInstance:=11788);
	RemoteControlStart_046: FB_BACnetRM_BV := (Client:=Client,nObjectInstance:=11789);
	
	RemoteControlTempAdjust_046: FB_BACnetRM_BV := (Client:=Client,nObjectInstance:=11792);
	
	
	
	
	
	
	
	
	
	
	
	
	//StartStopCommand_048: FB_BACnetRM_BO := (Client:=Client,nObjectInstance:=12289);
	//StartStopStatus_048: FB_BACnetRM_BI := (Client:=Client,nObjectInstance:=12290);
	//Alarm_048: FB_BACnetRM_BI := (Client:=Client,nObjectInstance:=12291);
	//MalfunctionCode_048: FB_BACnetRM_MI := (Client:=Client,nObjectInstance:=12292);
	
	
	
	
	//RoomTemp_048: FB_BACnetRM_AI := (Client:=Client,nObjectInstance:=12297);
	//TempAdjust_048: FB_BACnetRM_AV := (Client:=Client,nObjectInstance:=12298);
	//FilterSign_048: FB_BACnetRM_BI := (Client:=Client,nObjectInstance:=12299);
	//FilterSignReset_048: FB_BACnetRM_BV := (Client:=Client,nObjectInstance:=12300);
	//RemoteControlStart_048: FB_BACnetRM_BV := (Client:=Client,nObjectInstance:=12301);
	//
	//RemoteControlTempAdjust_048: FB_BACnetRM_BV := (Client:=Client,nObjectInstance:=12304);
	
	//
	
	
	
	
	
	
	
	
	
	
	StartStopCommand_049: FB_BACnetRM_BO := (Client:=Client,nObjectInstance:=12545);
	StartStopStatus_049: FB_BACnetRM_BI := (Client:=Client,nObjectInstance:=12546);
	Alarm_049: FB_BACnetRM_BI := (Client:=Client,nObjectInstance:=12547);
	MalfunctionCode_049: FB_BACnetRM_MI := (Client:=Client,nObjectInstance:=12548);
	
	
	
	
	RoomTemp_049: FB_BACnetRM_AI := (Client:=Client,nObjectInstance:=12553);
	TempAdjust_049: FB_BACnetRM_AV := (Client:=Client,nObjectInstance:=12554);
	FilterSign_049: FB_BACnetRM_BI := (Client:=Client,nObjectInstance:=12555);
	FilterSignReset_049: FB_BACnetRM_BV := (Client:=Client,nObjectInstance:=12556);
	RemoteControlStart_049: FB_BACnetRM_BV := (Client:=Client,nObjectInstance:=12557);
	
	RemoteControlTempAdjust_049: FB_BACnetRM_BV := (Client:=Client,nObjectInstance:=12560);
	
	
	
	
	
	
	
	
	
	
	
	
	StartStopCommand_064: FB_BACnetRM_BO := (Client:=Client,nObjectInstance:=16385);
	StartStopStatus_064: FB_BACnetRM_BI := (Client:=Client,nObjectInstance:=16386);
	Alarm_064: FB_BACnetRM_BI := (Client:=Client,nObjectInstance:=16387);
	MalfunctionCode_064: FB_BACnetRM_MI := (Client:=Client,nObjectInstance:=16388);
	
	
	
	
	RoomTemp_064: FB_BACnetRM_AI := (Client:=Client,nObjectInstance:=16393);
	TempAdjust_064: FB_BACnetRM_AV := (Client:=Client,nObjectInstance:=16394);
	FilterSign_064: FB_BACnetRM_BI := (Client:=Client,nObjectInstance:=16395);
	FilterSignReset_064: FB_BACnetRM_BV := (Client:=Client,nObjectInstance:=16396);
	RemoteControlStart_064: FB_BACnetRM_BV := (Client:=Client,nObjectInstance:=16397);
	
	RemoteControlTempAdjust_064: FB_BACnetRM_BV := (Client:=Client,nObjectInstance:=16400);
	
	
	
	
	
	
	
	
	
	
	
	
	StartStopCommand_065: FB_BACnetRM_BO := (Client:=Client,nObjectInstance:=16641);
	StartStopStatus_065: FB_BACnetRM_BI := (Client:=Client,nObjectInstance:=16642);
	Alarm_065: FB_BACnetRM_BI := (Client:=Client,nObjectInstance:=16643);
	MalfunctionCode_065: FB_BACnetRM_MI := (Client:=Client,nObjectInstance:=16644);
	
	
	
	
	RoomTemp_065: FB_BACnetRM_AI := (Client:=Client,nObjectInstance:=16649);
	TempAdjust_065: FB_BACnetRM_AV := (Client:=Client,nObjectInstance:=16650);
	FilterSign_065: FB_BACnetRM_BI := (Client:=Client,nObjectInstance:=16651);
	FilterSignReset_065: FB_BACnetRM_BV := (Client:=Client,nObjectInstance:=16652);
	RemoteControlStart_065: FB_BACnetRM_BV := (Client:=Client,nObjectInstance:=16653);
	
	RemoteControlTempAdjust_065: FB_BACnetRM_BV := (Client:=Client,nObjectInstance:=16656);
	
	
	
	
	
	
	
	
	
	
	
	
	StartStopCommand_066: FB_BACnetRM_BO := (Client:=Client,nObjectInstance:=16897);
	StartStopStatus_066: FB_BACnetRM_BI := (Client:=Client,nObjectInstance:=16898);
	Alarm_066: FB_BACnetRM_BI := (Client:=Client,nObjectInstance:=16899);
	MalfunctionCode_066: FB_BACnetRM_MI := (Client:=Client,nObjectInstance:=16900);
	
	
	
	
	RoomTemp_066: FB_BACnetRM_AI := (Client:=Client,nObjectInstance:=16905);
	TempAdjust_066: FB_BACnetRM_AV := (Client:=Client,nObjectInstance:=16906);
	FilterSign_066: FB_BACnetRM_BI := (Client:=Client,nObjectInstance:=16907);
	FilterSignReset_066: FB_BACnetRM_BV := (Client:=Client,nObjectInstance:=16908);
	RemoteControlStart_066: FB_BACnetRM_BV := (Client:=Client,nObjectInstance:=16909);
	
	RemoteControlTempAdjust_066: FB_BACnetRM_BV := (Client:=Client,nObjectInstance:=16912);
	
	
	
	
	
	
	
	
	
	
	
	
	StartStopCommand_067: FB_BACnetRM_BO := (Client:=Client,nObjectInstance:=17153);
	StartStopStatus_067: FB_BACnetRM_BI := (Client:=Client,nObjectInstance:=17154);
	Alarm_067: FB_BACnetRM_BI := (Client:=Client,nObjectInstance:=17155);
	MalfunctionCode_067: FB_BACnetRM_MI := (Client:=Client,nObjectInstance:=17156);
	
	
	
	
	RoomTemp_067: FB_BACnetRM_AI := (Client:=Client,nObjectInstance:=17161);
	TempAdjust_067: FB_BACnetRM_AV := (Client:=Client,nObjectInstance:=17162);
	FilterSign_067: FB_BACnetRM_BI := (Client:=Client,nObjectInstance:=17163);
	FilterSignReset_067: FB_BACnetRM_BV := (Client:=Client,nObjectInstance:=17164);
	RemoteControlStart_067: FB_BACnetRM_BV := (Client:=Client,nObjectInstance:=17165);
	
	RemoteControlTempAdjust_067: FB_BACnetRM_BV := (Client:=Client,nObjectInstance:=17168);
	
	
	
	
	
	
	
	
	
	
	
	
	StartStopCommand_068: FB_BACnetRM_BO := (Client:=Client,nObjectInstance:=17409);
	StartStopStatus_068: FB_BACnetRM_BI := (Client:=Client,nObjectInstance:=17410);
	Alarm_068: FB_BACnetRM_BI := (Client:=Client,nObjectInstance:=17411);
	MalfunctionCode_068: FB_BACnetRM_MI := (Client:=Client,nObjectInstance:=17412);
	
	
	
	
	RoomTemp_068: FB_BACnetRM_AI := (Client:=Client,nObjectInstance:=17417);
	TempAdjust_068: FB_BACnetRM_AV := (Client:=Client,nObjectInstance:=17418);
	FilterSign_068: FB_BACnetRM_BI := (Client:=Client,nObjectInstance:=17419);
	FilterSignReset_068: FB_BACnetRM_BV := (Client:=Client,nObjectInstance:=17420);
	RemoteControlStart_068: FB_BACnetRM_BV := (Client:=Client,nObjectInstance:=17421);
	
	RemoteControlTempAdjust_068: FB_BACnetRM_BV := (Client:=Client,nObjectInstance:=17424);
	
	
	
	
	
	
	
	
	
	
	
	
	StartStopCommand_069: FB_BACnetRM_BO := (Client:=Client,nObjectInstance:=17665);
	StartStopStatus_069: FB_BACnetRM_BI := (Client:=Client,nObjectInstance:=17666);
	Alarm_069: FB_BACnetRM_BI := (Client:=Client,nObjectInstance:=17667);
	MalfunctionCode_069: FB_BACnetRM_MI := (Client:=Client,nObjectInstance:=17668);
	
	
	
	
	RoomTemp_069: FB_BACnetRM_AI := (Client:=Client,nObjectInstance:=17673);
	TempAdjust_069: FB_BACnetRM_AV := (Client:=Client,nObjectInstance:=17674);
	FilterSign_069: FB_BACnetRM_BI := (Client:=Client,nObjectInstance:=17675);
	FilterSignReset_069: FB_BACnetRM_BV := (Client:=Client,nObjectInstance:=17676);
	RemoteControlStart_069: FB_BACnetRM_BV := (Client:=Client,nObjectInstance:=17677);
	
	RemoteControlTempAdjust_069: FB_BACnetRM_BV := (Client:=Client,nObjectInstance:=17680);
	
	
	
	
	
	
	
	
	
	
	
	
	StartStopCommand_070: FB_BACnetRM_BO := (Client:=Client,nObjectInstance:=17921);
	StartStopStatus_070: FB_BACnetRM_BI := (Client:=Client,nObjectInstance:=17922);
	Alarm_070: FB_BACnetRM_BI := (Client:=Client,nObjectInstance:=17923);
	MalfunctionCode_070: FB_BACnetRM_MI := (Client:=Client,nObjectInstance:=17924);
	
	
	
	
	RoomTemp_070: FB_BACnetRM_AI := (Client:=Client,nObjectInstance:=17929);
	TempAdjust_070: FB_BACnetRM_AV := (Client:=Client,nObjectInstance:=17930);
	FilterSign_070: FB_BACnetRM_BI := (Client:=Client,nObjectInstance:=17931);
	FilterSignReset_070: FB_BACnetRM_BV := (Client:=Client,nObjectInstance:=17932);
	RemoteControlStart_070: FB_BACnetRM_BV := (Client:=Client,nObjectInstance:=17933);
	
	RemoteControlTempAdjust_070: FB_BACnetRM_BV := (Client:=Client,nObjectInstance:=17936);
	
	
	
	
	
	
	
	
	
	
	
	
	StartStopCommand_071: FB_BACnetRM_BO := (Client:=Client,nObjectInstance:=18177);
	StartStopStatus_071: FB_BACnetRM_BI := (Client:=Client,nObjectInstance:=18178);
	Alarm_071: FB_BACnetRM_BI := (Client:=Client,nObjectInstance:=18179);
	MalfunctionCode_071: FB_BACnetRM_MI := (Client:=Client,nObjectInstance:=18180);
	
	
	
	
	RoomTemp_071: FB_BACnetRM_AI := (Client:=Client,nObjectInstance:=18185);
	TempAdjust_071: FB_BACnetRM_AV := (Client:=Client,nObjectInstance:=18186);
	FilterSign_071: FB_BACnetRM_BI := (Client:=Client,nObjectInstance:=18187);
	FilterSignReset_071: FB_BACnetRM_BV := (Client:=Client,nObjectInstance:=18188);
	RemoteControlStart_071: FB_BACnetRM_BV := (Client:=Client,nObjectInstance:=18189);
	
	RemoteControlTempAdjust_071: FB_BACnetRM_BV := (Client:=Client,nObjectInstance:=18192);
	
	
	
	
	
	
	
	
	
	
	
	
	StartStopCommand_072: FB_BACnetRM_BO := (Client:=Client,nObjectInstance:=18433);
	StartStopStatus_072: FB_BACnetRM_BI := (Client:=Client,nObjectInstance:=18434);
	Alarm_072: FB_BACnetRM_BI := (Client:=Client,nObjectInstance:=18435);
	MalfunctionCode_072: FB_BACnetRM_MI := (Client:=Client,nObjectInstance:=18436);
	
	
	
	
	RoomTemp_072: FB_BACnetRM_AI := (Client:=Client,nObjectInstance:=18441);
	TempAdjust_072: FB_BACnetRM_AV := (Client:=Client,nObjectInstance:=18442);
	FilterSign_072: FB_BACnetRM_BI := (Client:=Client,nObjectInstance:=18443);
	FilterSignReset_072: FB_BACnetRM_BV := (Client:=Client,nObjectInstance:=18444);
	RemoteControlStart_072: FB_BACnetRM_BV := (Client:=Client,nObjectInstance:=18445);
	
	RemoteControlTempAdjust_072: FB_BACnetRM_BV := (Client:=Client,nObjectInstance:=18448);
	
	
	
	
	
	
	
	
	
	
	
	
	StartStopCommand_073: FB_BACnetRM_BO := (Client:=Client,nObjectInstance:=18689);
	StartStopStatus_073: FB_BACnetRM_BI := (Client:=Client,nObjectInstance:=18690);
	Alarm_073: FB_BACnetRM_BI := (Client:=Client,nObjectInstance:=18691);
	MalfunctionCode_073: FB_BACnetRM_MI := (Client:=Client,nObjectInstance:=18692);
	
	
	
	
	RoomTemp_073: FB_BACnetRM_AI := (Client:=Client,nObjectInstance:=18697);
	TempAdjust_073: FB_BACnetRM_AV := (Client:=Client,nObjectInstance:=18698);
	FilterSign_073: FB_BACnetRM_BI := (Client:=Client,nObjectInstance:=18699);
	FilterSignReset_073: FB_BACnetRM_BV := (Client:=Client,nObjectInstance:=18700);
	RemoteControlStart_073: FB_BACnetRM_BV := (Client:=Client,nObjectInstance:=18701);
	
	RemoteControlTempAdjust_073: FB_BACnetRM_BV := (Client:=Client,nObjectInstance:=18704);
	
	
	
	
	
	
	
	
	
	
	
	
	StartStopCommand_074: FB_BACnetRM_BO := (Client:=Client,nObjectInstance:=18945);
	StartStopStatus_074: FB_BACnetRM_BI := (Client:=Client,nObjectInstance:=18946);
	Alarm_074: FB_BACnetRM_BI := (Client:=Client,nObjectInstance:=18947);
	MalfunctionCode_074: FB_BACnetRM_MI := (Client:=Client,nObjectInstance:=18948);
	
	
	
	
	RoomTemp_074: FB_BACnetRM_AI := (Client:=Client,nObjectInstance:=18953);
	TempAdjust_074: FB_BACnetRM_AV := (Client:=Client,nObjectInstance:=18954);
	FilterSign_074: FB_BACnetRM_BI := (Client:=Client,nObjectInstance:=18955);
	FilterSignReset_074: FB_BACnetRM_BV := (Client:=Client,nObjectInstance:=18956);
	RemoteControlStart_074: FB_BACnetRM_BV := (Client:=Client,nObjectInstance:=18957);
	
	RemoteControlTempAdjust_074: FB_BACnetRM_BV := (Client:=Client,nObjectInstance:=18960);
	
	
	
	
	
	
	
	
	
	
	
	
	StartStopCommand_075: FB_BACnetRM_BO := (Client:=Client,nObjectInstance:=19201);
	StartStopStatus_075: FB_BACnetRM_BI := (Client:=Client,nObjectInstance:=19202);
	Alarm_075: FB_BACnetRM_BI := (Client:=Client,nObjectInstance:=19203);
	MalfunctionCode_075: FB_BACnetRM_MI := (Client:=Client,nObjectInstance:=19204);
	
	
	
	
	RoomTemp_075: FB_BACnetRM_AI := (Client:=Client,nObjectInstance:=19209);
	TempAdjust_075: FB_BACnetRM_AV := (Client:=Client,nObjectInstance:=19210);
	FilterSign_075: FB_BACnetRM_BI := (Client:=Client,nObjectInstance:=19211);
	FilterSignReset_075: FB_BACnetRM_BV := (Client:=Client,nObjectInstance:=19212);
	RemoteControlStart_075: FB_BACnetRM_BV := (Client:=Client,nObjectInstance:=19213);
	
	RemoteControlTempAdjust_075: FB_BACnetRM_BV := (Client:=Client,nObjectInstance:=19216);
	
	
	
	
	
	
	
	
	
	
	
	
	StartStopCommand_076: FB_BACnetRM_BO := (Client:=Client,nObjectInstance:=19457);
	StartStopStatus_076: FB_BACnetRM_BI := (Client:=Client,nObjectInstance:=19458);
	Alarm_076: FB_BACnetRM_BI := (Client:=Client,nObjectInstance:=19459);
	MalfunctionCode_076: FB_BACnetRM_MI := (Client:=Client,nObjectInstance:=19460);
	
	
	
	
	RoomTemp_076: FB_BACnetRM_AI := (Client:=Client,nObjectInstance:=19465);
	TempAdjust_076: FB_BACnetRM_AV := (Client:=Client,nObjectInstance:=19466);
	FilterSign_076: FB_BACnetRM_BI := (Client:=Client,nObjectInstance:=19467);
	FilterSignReset_076: FB_BACnetRM_BV := (Client:=Client,nObjectInstance:=19468);
	RemoteControlStart_076: FB_BACnetRM_BV := (Client:=Client,nObjectInstance:=19469);
	
	RemoteControlTempAdjust_076: FB_BACnetRM_BV := (Client:=Client,nObjectInstance:=19472);
	
	
	
	
	
	
	
	
	
	
	
	
	StartStopCommand_077: FB_BACnetRM_BO := (Client:=Client,nObjectInstance:=19713);
	StartStopStatus_077: FB_BACnetRM_BI := (Client:=Client,nObjectInstance:=19714);
	Alarm_077: FB_BACnetRM_BI := (Client:=Client,nObjectInstance:=19715);
	MalfunctionCode_077: FB_BACnetRM_MI := (Client:=Client,nObjectInstance:=19716);
	
	
	
	
	RoomTemp_077: FB_BACnetRM_AI := (Client:=Client,nObjectInstance:=19721);
	TempAdjust_077: FB_BACnetRM_AV := (Client:=Client,nObjectInstance:=19722);
	FilterSign_077: FB_BACnetRM_BI := (Client:=Client,nObjectInstance:=19723);
	FilterSignReset_077: FB_BACnetRM_BV := (Client:=Client,nObjectInstance:=19724);
	RemoteControlStart_077: FB_BACnetRM_BV := (Client:=Client,nObjectInstance:=19725);
	
	RemoteControlTempAdjust_077: FB_BACnetRM_BV := (Client:=Client,nObjectInstance:=19728);
	
	
	
	
	
	
	
	
	
	
	
	
	StartStopCommand_078: FB_BACnetRM_BO := (Client:=Client,nObjectInstance:=19969);
	StartStopStatus_078: FB_BACnetRM_BI := (Client:=Client,nObjectInstance:=19970);
	Alarm_078: FB_BACnetRM_BI := (Client:=Client,nObjectInstance:=19971);
	MalfunctionCode_078: FB_BACnetRM_MI := (Client:=Client,nObjectInstance:=19972);
	
	
	
	
	RoomTemp_078: FB_BACnetRM_AI := (Client:=Client,nObjectInstance:=19977);
	TempAdjust_078: FB_BACnetRM_AV := (Client:=Client,nObjectInstance:=19978);
	FilterSign_078: FB_BACnetRM_BI := (Client:=Client,nObjectInstance:=19979);
	FilterSignReset_078: FB_BACnetRM_BV := (Client:=Client,nObjectInstance:=19980);
	RemoteControlStart_078: FB_BACnetRM_BV := (Client:=Client,nObjectInstance:=19981);
	
	RemoteControlTempAdjust_078: FB_BACnetRM_BV := (Client:=Client,nObjectInstance:=19984);
	
	
	
	
	
	
	
	
	
	
	
	
	StartStopCommand_079: FB_BACnetRM_BO := (Client:=Client,nObjectInstance:=20225);
	StartStopStatus_079: FB_BACnetRM_BI := (Client:=Client,nObjectInstance:=20226);
	Alarm_079: FB_BACnetRM_BI := (Client:=Client,nObjectInstance:=20227);
	MalfunctionCode_079: FB_BACnetRM_MI := (Client:=Client,nObjectInstance:=20228);
	
	
	
	
	RoomTemp_079: FB_BACnetRM_AI := (Client:=Client,nObjectInstance:=20233);
	TempAdjust_079: FB_BACnetRM_AV := (Client:=Client,nObjectInstance:=20234);
	FilterSign_079: FB_BACnetRM_BI := (Client:=Client,nObjectInstance:=20235);
	FilterSignReset_079: FB_BACnetRM_BV := (Client:=Client,nObjectInstance:=20236);
	RemoteControlStart_079: FB_BACnetRM_BV := (Client:=Client,nObjectInstance:=20237);
	
	RemoteControlTempAdjust_079: FB_BACnetRM_BV := (Client:=Client,nObjectInstance:=20240);
	
	
	
	
	
	
	
	
	
	
	
	
	StartStopCommand_080: FB_BACnetRM_BO := (Client:=Client,nObjectInstance:=20481);
	StartStopStatus_080: FB_BACnetRM_BI := (Client:=Client,nObjectInstance:=20482);
	Alarm_080: FB_BACnetRM_BI := (Client:=Client,nObjectInstance:=20483);
	MalfunctionCode_080: FB_BACnetRM_MI := (Client:=Client,nObjectInstance:=20484);
	
	
	
	
	RoomTemp_080: FB_BACnetRM_AI := (Client:=Client,nObjectInstance:=20489);
	TempAdjust_080: FB_BACnetRM_AV := (Client:=Client,nObjectInstance:=20490);
	FilterSign_080: FB_BACnetRM_BI := (Client:=Client,nObjectInstance:=20491);
	FilterSignReset_080: FB_BACnetRM_BV := (Client:=Client,nObjectInstance:=20492);
	RemoteControlStart_080: FB_BACnetRM_BV := (Client:=Client,nObjectInstance:=20493);
	
	RemoteControlTempAdjust_080: FB_BACnetRM_BV := (Client:=Client,nObjectInstance:=20496);
	
	
	
	
	
	
	
	
	
	
	
	
	StartStopCommand_081: FB_BACnetRM_BO := (Client:=Client,nObjectInstance:=20737);
	StartStopStatus_081: FB_BACnetRM_BI := (Client:=Client,nObjectInstance:=20738);
	Alarm_081: FB_BACnetRM_BI := (Client:=Client,nObjectInstance:=20739);
	MalfunctionCode_081: FB_BACnetRM_MI := (Client:=Client,nObjectInstance:=20740);
	
	
	
	
	RoomTemp_081: FB_BACnetRM_AI := (Client:=Client,nObjectInstance:=20745);
	TempAdjust_081: FB_BACnetRM_AV := (Client:=Client,nObjectInstance:=20746);
	FilterSign_081: FB_BACnetRM_BI := (Client:=Client,nObjectInstance:=20747);
	FilterSignReset_081: FB_BACnetRM_BV := (Client:=Client,nObjectInstance:=20748);
	RemoteControlStart_081: FB_BACnetRM_BV := (Client:=Client,nObjectInstance:=20749);
	
	RemoteControlTempAdjust_081: FB_BACnetRM_BV := (Client:=Client,nObjectInstance:=20752);
	
	
	
	
	
	
	
	
	
	
	
	
	StartStopCommand_082: FB_BACnetRM_BO := (Client:=Client,nObjectInstance:=20993);
	StartStopStatus_082: FB_BACnetRM_BI := (Client:=Client,nObjectInstance:=20994);
	Alarm_082: FB_BACnetRM_BI := (Client:=Client,nObjectInstance:=20995);
	MalfunctionCode_082: FB_BACnetRM_MI := (Client:=Client,nObjectInstance:=20996);
	
	
	
	
	RoomTemp_082: FB_BACnetRM_AI := (Client:=Client,nObjectInstance:=21001);
	TempAdjust_082: FB_BACnetRM_AV := (Client:=Client,nObjectInstance:=21002);
	FilterSign_082: FB_BACnetRM_BI := (Client:=Client,nObjectInstance:=21003);
	FilterSignReset_082: FB_BACnetRM_BV := (Client:=Client,nObjectInstance:=21004);
	RemoteControlStart_082: FB_BACnetRM_BV := (Client:=Client,nObjectInstance:=21005);
	
	RemoteControlTempAdjust_082: FB_BACnetRM_BV := (Client:=Client,nObjectInstance:=21008);
	
	
	
	
	
	
	
	
	
	
	
	
	StartStopCommand_083: FB_BACnetRM_BO := (Client:=Client,nObjectInstance:=21249);
	StartStopStatus_083: FB_BACnetRM_BI := (Client:=Client,nObjectInstance:=21250);
	Alarm_083: FB_BACnetRM_BI := (Client:=Client,nObjectInstance:=21251);
	MalfunctionCode_083: FB_BACnetRM_MI := (Client:=Client,nObjectInstance:=21252);
	
	
	
	
	RoomTemp_083: FB_BACnetRM_AI := (Client:=Client,nObjectInstance:=21257);
	TempAdjust_083: FB_BACnetRM_AV := (Client:=Client,nObjectInstance:=21258);
	FilterSign_083: FB_BACnetRM_BI := (Client:=Client,nObjectInstance:=21259);
	FilterSignReset_083: FB_BACnetRM_BV := (Client:=Client,nObjectInstance:=21260);
	RemoteControlStart_083: FB_BACnetRM_BV := (Client:=Client,nObjectInstance:=21261);
	
	RemoteControlTempAdjust_083: FB_BACnetRM_BV := (Client:=Client,nObjectInstance:=21264);
	
	
	
	
	
	
	
	
	
	
	
	
	StartStopCommand_084: FB_BACnetRM_BO := (Client:=Client,nObjectInstance:=21505);
	StartStopStatus_084: FB_BACnetRM_BI := (Client:=Client,nObjectInstance:=21506);
	Alarm_084: FB_BACnetRM_BI := (Client:=Client,nObjectInstance:=21507);
	MalfunctionCode_084: FB_BACnetRM_MI := (Client:=Client,nObjectInstance:=21508);
	
	
	
	
	RoomTemp_084: FB_BACnetRM_AI := (Client:=Client,nObjectInstance:=21513);
	TempAdjust_084: FB_BACnetRM_AV := (Client:=Client,nObjectInstance:=21514);
	FilterSign_084: FB_BACnetRM_BI := (Client:=Client,nObjectInstance:=21515);
	FilterSignReset_084: FB_BACnetRM_BV := (Client:=Client,nObjectInstance:=21516);
	RemoteControlStart_084: FB_BACnetRM_BV := (Client:=Client,nObjectInstance:=21517);
	
	RemoteControlTempAdjust_084: FB_BACnetRM_BV := (Client:=Client,nObjectInstance:=21520);
	
	
	
	
	
	
	
	
	
	
	
	
	StartStopCommand_085: FB_BACnetRM_BO := (Client:=Client,nObjectInstance:=21761);
	StartStopStatus_085: FB_BACnetRM_BI := (Client:=Client,nObjectInstance:=21762);
	Alarm_085: FB_BACnetRM_BI := (Client:=Client,nObjectInstance:=21763);
	MalfunctionCode_085: FB_BACnetRM_MI := (Client:=Client,nObjectInstance:=21764);
	
	
	
	
	RoomTemp_085: FB_BACnetRM_AI := (Client:=Client,nObjectInstance:=21769);
	TempAdjust_085: FB_BACnetRM_AV := (Client:=Client,nObjectInstance:=21770);
	FilterSign_085: FB_BACnetRM_BI := (Client:=Client,nObjectInstance:=21771);
	FilterSignReset_085: FB_BACnetRM_BV := (Client:=Client,nObjectInstance:=21772);
	RemoteControlStart_085: FB_BACnetRM_BV := (Client:=Client,nObjectInstance:=21773);
	
	RemoteControlTempAdjust_085: FB_BACnetRM_BV := (Client:=Client,nObjectInstance:=21776);
	
	
	
	
	
	
	
	
	
	
	
	
	StartStopCommand_096: FB_BACnetRM_BO := (Client:=Client,nObjectInstance:=24577);
	StartStopStatus_096: FB_BACnetRM_BI := (Client:=Client,nObjectInstance:=24578);
	Alarm_096: FB_BACnetRM_BI := (Client:=Client,nObjectInstance:=24579);
	MalfunctionCode_096: FB_BACnetRM_MI := (Client:=Client,nObjectInstance:=24580);
	
	
	
	
	RoomTemp_096: FB_BACnetRM_AI := (Client:=Client,nObjectInstance:=24585);
	TempAdjust_096: FB_BACnetRM_AV := (Client:=Client,nObjectInstance:=24586);
	FilterSign_096: FB_BACnetRM_BI := (Client:=Client,nObjectInstance:=24587);
	FilterSignReset_096: FB_BACnetRM_BV := (Client:=Client,nObjectInstance:=24588);
	RemoteControlStart_096: FB_BACnetRM_BV := (Client:=Client,nObjectInstance:=24589);
	
	RemoteControlTempAdjust_096: FB_BACnetRM_BV := (Client:=Client,nObjectInstance:=24592);
	
	
	
	
	
	
	
	
	
	
	
	
	StartStopCommand_097: FB_BACnetRM_BO := (Client:=Client,nObjectInstance:=24833);
	StartStopStatus_097: FB_BACnetRM_BI := (Client:=Client,nObjectInstance:=24834);
	Alarm_097: FB_BACnetRM_BI := (Client:=Client,nObjectInstance:=24835);
	MalfunctionCode_097: FB_BACnetRM_MI := (Client:=Client,nObjectInstance:=24836);
	
	
	
	
	RoomTemp_097: FB_BACnetRM_AI := (Client:=Client,nObjectInstance:=24841);
	TempAdjust_097: FB_BACnetRM_AV := (Client:=Client,nObjectInstance:=24842);
	FilterSign_097: FB_BACnetRM_BI := (Client:=Client,nObjectInstance:=24843);
	FilterSignReset_097: FB_BACnetRM_BV := (Client:=Client,nObjectInstance:=24844);
	RemoteControlStart_097: FB_BACnetRM_BV := (Client:=Client,nObjectInstance:=24845);
	
	RemoteControlTempAdjust_097: FB_BACnetRM_BV := (Client:=Client,nObjectInstance:=24848);
	
	
	
	
	
	
	
	
	
	
	
	
	StartStopCommand_098: FB_BACnetRM_BO := (Client:=Client,nObjectInstance:=25089);
	StartStopStatus_098: FB_BACnetRM_BI := (Client:=Client,nObjectInstance:=25090);
	Alarm_098: FB_BACnetRM_BI := (Client:=Client,nObjectInstance:=25091);
	MalfunctionCode_098: FB_BACnetRM_MI := (Client:=Client,nObjectInstance:=25092);
	
	
	
	
	RoomTemp_098: FB_BACnetRM_AI := (Client:=Client,nObjectInstance:=25097);
	TempAdjust_098: FB_BACnetRM_AV := (Client:=Client,nObjectInstance:=25098);
	FilterSign_098: FB_BACnetRM_BI := (Client:=Client,nObjectInstance:=25099);
	FilterSignReset_098: FB_BACnetRM_BV := (Client:=Client,nObjectInstance:=25100);
	RemoteControlStart_098: FB_BACnetRM_BV := (Client:=Client,nObjectInstance:=25101);
	
	RemoteControlTempAdjust_098: FB_BACnetRM_BV := (Client:=Client,nObjectInstance:=25104);
	
	
	
	
	
	
	
	
	
	
	
	
	StartStopCommand_099: FB_BACnetRM_BO := (Client:=Client,nObjectInstance:=25345);
	StartStopStatus_099: FB_BACnetRM_BI := (Client:=Client,nObjectInstance:=25346);
	Alarm_099: FB_BACnetRM_BI := (Client:=Client,nObjectInstance:=25347);
	MalfunctionCode_099: FB_BACnetRM_MI := (Client:=Client,nObjectInstance:=25348);
	
	
	
	
	RoomTemp_099: FB_BACnetRM_AI := (Client:=Client,nObjectInstance:=25353);
	TempAdjust_099: FB_BACnetRM_AV := (Client:=Client,nObjectInstance:=25354);
	FilterSign_099: FB_BACnetRM_BI := (Client:=Client,nObjectInstance:=25355);
	FilterSignReset_099: FB_BACnetRM_BV := (Client:=Client,nObjectInstance:=25356);
	RemoteControlStart_099: FB_BACnetRM_BV := (Client:=Client,nObjectInstance:=25357);
	
	RemoteControlTempAdjust_099: FB_BACnetRM_BV := (Client:=Client,nObjectInstance:=25360);
	
	
	
	
	
	
	
	
	
	
	
	
	StartStopCommand_100: FB_BACnetRM_BO := (Client:=Client,nObjectInstance:=25601);
	StartStopStatus_100: FB_BACnetRM_BI := (Client:=Client,nObjectInstance:=25602);
	Alarm_100: FB_BACnetRM_BI := (Client:=Client,nObjectInstance:=25603);
	MalfunctionCode_100: FB_BACnetRM_MI := (Client:=Client,nObjectInstance:=25604);
	
	
	
	
	RoomTemp_100: FB_BACnetRM_AI := (Client:=Client,nObjectInstance:=25609);
	TempAdjust_100: FB_BACnetRM_AV := (Client:=Client,nObjectInstance:=25610);
	FilterSign_100: FB_BACnetRM_BI := (Client:=Client,nObjectInstance:=25611);
	FilterSignReset_100: FB_BACnetRM_BV := (Client:=Client,nObjectInstance:=25612);
	RemoteControlStart_100: FB_BACnetRM_BV := (Client:=Client,nObjectInstance:=25613);
	
	RemoteControlTempAdjust_100: FB_BACnetRM_BV := (Client:=Client,nObjectInstance:=25616);
	
	
	
	
	
	
	
	
	
	
	
	
	StartStopCommand_101: FB_BACnetRM_BO := (Client:=Client,nObjectInstance:=25857);
	StartStopStatus_101: FB_BACnetRM_BI := (Client:=Client,nObjectInstance:=25858);
	Alarm_101: FB_BACnetRM_BI := (Client:=Client,nObjectInstance:=25859);
	MalfunctionCode_101: FB_BACnetRM_MI := (Client:=Client,nObjectInstance:=25860);
	
	
	
	
	RoomTemp_101: FB_BACnetRM_AI := (Client:=Client,nObjectInstance:=25865);
	TempAdjust_101: FB_BACnetRM_AV := (Client:=Client,nObjectInstance:=25866);
	FilterSign_101: FB_BACnetRM_BI := (Client:=Client,nObjectInstance:=25867);
	FilterSignReset_101: FB_BACnetRM_BV := (Client:=Client,nObjectInstance:=25868);
	RemoteControlStart_101: FB_BACnetRM_BV := (Client:=Client,nObjectInstance:=25869);
	
	RemoteControlTempAdjust_101: FB_BACnetRM_BV := (Client:=Client,nObjectInstance:=25872);
	
	
	
	
	
	
	
	
	
	
	
	
	StartStopCommand_102: FB_BACnetRM_BO := (Client:=Client,nObjectInstance:=26113);
	StartStopStatus_102: FB_BACnetRM_BI := (Client:=Client,nObjectInstance:=26114);
	Alarm_102: FB_BACnetRM_BI := (Client:=Client,nObjectInstance:=26115);
	MalfunctionCode_102: FB_BACnetRM_MI := (Client:=Client,nObjectInstance:=26116);
	
	
	
	
	RoomTemp_102: FB_BACnetRM_AI := (Client:=Client,nObjectInstance:=26121);
	TempAdjust_102: FB_BACnetRM_AV := (Client:=Client,nObjectInstance:=26122);
	FilterSign_102: FB_BACnetRM_BI := (Client:=Client,nObjectInstance:=26123);
	FilterSignReset_102: FB_BACnetRM_BV := (Client:=Client,nObjectInstance:=26124);
	RemoteControlStart_102: FB_BACnetRM_BV := (Client:=Client,nObjectInstance:=26125);
	
	RemoteControlTempAdjust_102: FB_BACnetRM_BV := (Client:=Client,nObjectInstance:=26128);
	
	
	
	
	
	
	
	
	
	
	
	
	StartStopCommand_103: FB_BACnetRM_BO := (Client:=Client,nObjectInstance:=26369);
	StartStopStatus_103: FB_BACnetRM_BI := (Client:=Client,nObjectInstance:=26370);
	Alarm_103: FB_BACnetRM_BI := (Client:=Client,nObjectInstance:=26371);
	MalfunctionCode_103: FB_BACnetRM_MI := (Client:=Client,nObjectInstance:=26372);
	
	
	
	
	RoomTemp_103: FB_BACnetRM_AI := (Client:=Client,nObjectInstance:=26377);
	TempAdjust_103: FB_BACnetRM_AV := (Client:=Client,nObjectInstance:=26378);
	FilterSign_103: FB_BACnetRM_BI := (Client:=Client,nObjectInstance:=26379);
	FilterSignReset_103: FB_BACnetRM_BV := (Client:=Client,nObjectInstance:=26380);
	RemoteControlStart_103: FB_BACnetRM_BV := (Client:=Client,nObjectInstance:=26381);
	
	RemoteControlTempAdjust_103: FB_BACnetRM_BV := (Client:=Client,nObjectInstance:=26384);
	
	
	
	
	
	
	
	
	
	
	
	
	StartStopCommand_104: FB_BACnetRM_BO := (Client:=Client,nObjectInstance:=26625);
	StartStopStatus_104: FB_BACnetRM_BI := (Client:=Client,nObjectInstance:=26626);
	Alarm_104: FB_BACnetRM_BI := (Client:=Client,nObjectInstance:=26627);
	MalfunctionCode_104: FB_BACnetRM_MI := (Client:=Client,nObjectInstance:=26628);
	
	
	
	
	RoomTemp_104: FB_BACnetRM_AI := (Client:=Client,nObjectInstance:=26633);
	TempAdjust_104: FB_BACnetRM_AV := (Client:=Client,nObjectInstance:=26634);
	FilterSign_104: FB_BACnetRM_BI := (Client:=Client,nObjectInstance:=26635);
	FilterSignReset_104: FB_BACnetRM_BV := (Client:=Client,nObjectInstance:=26636);
	RemoteControlStart_104: FB_BACnetRM_BV := (Client:=Client,nObjectInstance:=26637);
	
	RemoteControlTempAdjust_104: FB_BACnetRM_BV := (Client:=Client,nObjectInstance:=26640);
	
	
	
	
	
	
	
	
	
	
	
	
	StartStopCommand_105: FB_BACnetRM_BO := (Client:=Client,nObjectInstance:=26881);
	StartStopStatus_105: FB_BACnetRM_BI := (Client:=Client,nObjectInstance:=26882);
	Alarm_105: FB_BACnetRM_BI := (Client:=Client,nObjectInstance:=26883);
	MalfunctionCode_105: FB_BACnetRM_MI := (Client:=Client,nObjectInstance:=26884);
	
	
	
	
	RoomTemp_105: FB_BACnetRM_AI := (Client:=Client,nObjectInstance:=26889);
	TempAdjust_105: FB_BACnetRM_AV := (Client:=Client,nObjectInstance:=26890);
	FilterSign_105: FB_BACnetRM_BI := (Client:=Client,nObjectInstance:=26891);
	FilterSignReset_105: FB_BACnetRM_BV := (Client:=Client,nObjectInstance:=26892);
	RemoteControlStart_105: FB_BACnetRM_BV := (Client:=Client,nObjectInstance:=26893);
	
	RemoteControlTempAdjust_105: FB_BACnetRM_BV := (Client:=Client,nObjectInstance:=26896);
	
	
	
	
	
	
	
	
	
	
	
	
	StartStopCommand_128: FB_BACnetRM_BO := (Client:=Client,nObjectInstance:=32769);
	StartStopStatus_128: FB_BACnetRM_BI := (Client:=Client,nObjectInstance:=32770);
	Alarm_128: FB_BACnetRM_BI := (Client:=Client,nObjectInstance:=32771);
	MalfunctionCode_128: FB_BACnetRM_MI := (Client:=Client,nObjectInstance:=32772);
	
	
	
	
	RoomTemp_128: FB_BACnetRM_AI := (Client:=Client,nObjectInstance:=32777);
	TempAdjust_128: FB_BACnetRM_AV := (Client:=Client,nObjectInstance:=32778);
	FilterSign_128: FB_BACnetRM_BI := (Client:=Client,nObjectInstance:=32779);
	FilterSignReset_128: FB_BACnetRM_BV := (Client:=Client,nObjectInstance:=32780);
	RemoteControlStart_128: FB_BACnetRM_BV := (Client:=Client,nObjectInstance:=32781);
	
	RemoteControlTempAdjust_128: FB_BACnetRM_BV := (Client:=Client,nObjectInstance:=32784);
	
	
	
	
	
	
	
	
	
	
	
	
	StartStopCommand_129: FB_BACnetRM_BO := (Client:=Client,nObjectInstance:=33025);
	StartStopStatus_129: FB_BACnetRM_BI := (Client:=Client,nObjectInstance:=33026);
	Alarm_129: FB_BACnetRM_BI := (Client:=Client,nObjectInstance:=33027);
	MalfunctionCode_129: FB_BACnetRM_MI := (Client:=Client,nObjectInstance:=33028);
	
	
	
	
	RoomTemp_129: FB_BACnetRM_AI := (Client:=Client,nObjectInstance:=33033);
	TempAdjust_129: FB_BACnetRM_AV := (Client:=Client,nObjectInstance:=33034);
	FilterSign_129: FB_BACnetRM_BI := (Client:=Client,nObjectInstance:=33035);
	FilterSignReset_129: FB_BACnetRM_BV := (Client:=Client,nObjectInstance:=33036);
	RemoteControlStart_129: FB_BACnetRM_BV := (Client:=Client,nObjectInstance:=33037);
	
	RemoteControlTempAdjust_129: FB_BACnetRM_BV := (Client:=Client,nObjectInstance:=33040);
	
	
	
	
	
	
	
	
	
	
	
	
	StartStopCommand_130: FB_BACnetRM_BO := (Client:=Client,nObjectInstance:=33281);
	StartStopStatus_130: FB_BACnetRM_BI := (Client:=Client,nObjectInstance:=33282);
	Alarm_130: FB_BACnetRM_BI := (Client:=Client,nObjectInstance:=33283);
	MalfunctionCode_130: FB_BACnetRM_MI := (Client:=Client,nObjectInstance:=33284);
	
	
	
	
	RoomTemp_130: FB_BACnetRM_AI := (Client:=Client,nObjectInstance:=33289);
	TempAdjust_130: FB_BACnetRM_AV := (Client:=Client,nObjectInstance:=33290);
	FilterSign_130: FB_BACnetRM_BI := (Client:=Client,nObjectInstance:=33291);
	FilterSignReset_130: FB_BACnetRM_BV := (Client:=Client,nObjectInstance:=33292);
	RemoteControlStart_130: FB_BACnetRM_BV := (Client:=Client,nObjectInstance:=33293);
	
	RemoteControlTempAdjust_130: FB_BACnetRM_BV := (Client:=Client,nObjectInstance:=33296);
	
	
	
	
	
	
	
	
	
	
	
	
	StartStopCommand_131: FB_BACnetRM_BO := (Client:=Client,nObjectInstance:=33537);
	StartStopStatus_131: FB_BACnetRM_BI := (Client:=Client,nObjectInstance:=33538);
	Alarm_131: FB_BACnetRM_BI := (Client:=Client,nObjectInstance:=33539);
	MalfunctionCode_131: FB_BACnetRM_MI := (Client:=Client,nObjectInstance:=33540);
	
	
	
	
	RoomTemp_131: FB_BACnetRM_AI := (Client:=Client,nObjectInstance:=33545);
	TempAdjust_131: FB_BACnetRM_AV := (Client:=Client,nObjectInstance:=33546);
	FilterSign_131: FB_BACnetRM_BI := (Client:=Client,nObjectInstance:=33547);
	FilterSignReset_131: FB_BACnetRM_BV := (Client:=Client,nObjectInstance:=33548);
	RemoteControlStart_131: FB_BACnetRM_BV := (Client:=Client,nObjectInstance:=33549);
	
	RemoteControlTempAdjust_131: FB_BACnetRM_BV := (Client:=Client,nObjectInstance:=33552);
	
	
	
	
	
	
	
	
	
	
	
	
	StartStopCommand_132: FB_BACnetRM_BO := (Client:=Client,nObjectInstance:=33793);
	StartStopStatus_132: FB_BACnetRM_BI := (Client:=Client,nObjectInstance:=33794);
	Alarm_132: FB_BACnetRM_BI := (Client:=Client,nObjectInstance:=33795);
	MalfunctionCode_132: FB_BACnetRM_MI := (Client:=Client,nObjectInstance:=33796);
	
	
	
	
	RoomTemp_132: FB_BACnetRM_AI := (Client:=Client,nObjectInstance:=33801);
	TempAdjust_132: FB_BACnetRM_AV := (Client:=Client,nObjectInstance:=33802);
	FilterSign_132: FB_BACnetRM_BI := (Client:=Client,nObjectInstance:=33803);
	FilterSignReset_132: FB_BACnetRM_BV := (Client:=Client,nObjectInstance:=33804);
	RemoteControlStart_132: FB_BACnetRM_BV := (Client:=Client,nObjectInstance:=33805);
	
	RemoteControlTempAdjust_132: FB_BACnetRM_BV := (Client:=Client,nObjectInstance:=33808);
	
	
	
	
	
	
	
	
	
	
	
	
	StartStopCommand_133: FB_BACnetRM_BO := (Client:=Client,nObjectInstance:=34049);
	StartStopStatus_133: FB_BACnetRM_BI := (Client:=Client,nObjectInstance:=34050);
	Alarm_133: FB_BACnetRM_BI := (Client:=Client,nObjectInstance:=34051);
	MalfunctionCode_133: FB_BACnetRM_MI := (Client:=Client,nObjectInstance:=34052);
	
	
	
	
	RoomTemp_133: FB_BACnetRM_AI := (Client:=Client,nObjectInstance:=34057);
	TempAdjust_133: FB_BACnetRM_AV := (Client:=Client,nObjectInstance:=34058);
	FilterSign_133: FB_BACnetRM_BI := (Client:=Client,nObjectInstance:=34059);
	FilterSignReset_133: FB_BACnetRM_BV := (Client:=Client,nObjectInstance:=34060);
	RemoteControlStart_133: FB_BACnetRM_BV := (Client:=Client,nObjectInstance:=34061);
	
	RemoteControlTempAdjust_133: FB_BACnetRM_BV := (Client:=Client,nObjectInstance:=34064);
	
	
	
	
	
	
	
	
	
	
	
	
	StartStopCommand_134: FB_BACnetRM_BO := (Client:=Client,nObjectInstance:=34305);
	StartStopStatus_134: FB_BACnetRM_BI := (Client:=Client,nObjectInstance:=34306);
	Alarm_134: FB_BACnetRM_BI := (Client:=Client,nObjectInstance:=34307);
	MalfunctionCode_134: FB_BACnetRM_MI := (Client:=Client,nObjectInstance:=34308);
	
	
	
	
	RoomTemp_134: FB_BACnetRM_AI := (Client:=Client,nObjectInstance:=34313);
	TempAdjust_134: FB_BACnetRM_AV := (Client:=Client,nObjectInstance:=34314);
	FilterSign_134: FB_BACnetRM_BI := (Client:=Client,nObjectInstance:=34315);
	FilterSignReset_134: FB_BACnetRM_BV := (Client:=Client,nObjectInstance:=34316);
	RemoteControlStart_134: FB_BACnetRM_BV := (Client:=Client,nObjectInstance:=34317);
	
	RemoteControlTempAdjust_134: FB_BACnetRM_BV := (Client:=Client,nObjectInstance:=34320);
	
	
	
	
	
	
	
	
	
	
	
	
	StartStopCommand_135: FB_BACnetRM_BO := (Client:=Client,nObjectInstance:=34561);
	StartStopStatus_135: FB_BACnetRM_BI := (Client:=Client,nObjectInstance:=34562);
	Alarm_135: FB_BACnetRM_BI := (Client:=Client,nObjectInstance:=34563);
	MalfunctionCode_135: FB_BACnetRM_MI := (Client:=Client,nObjectInstance:=34564);
	
	
	
	
	RoomTemp_135: FB_BACnetRM_AI := (Client:=Client,nObjectInstance:=34569);
	TempAdjust_135: FB_BACnetRM_AV := (Client:=Client,nObjectInstance:=34570);
	FilterSign_135: FB_BACnetRM_BI := (Client:=Client,nObjectInstance:=34571);
	FilterSignReset_135: FB_BACnetRM_BV := (Client:=Client,nObjectInstance:=34572);
	RemoteControlStart_135: FB_BACnetRM_BV := (Client:=Client,nObjectInstance:=34573);
	
	RemoteControlTempAdjust_135: FB_BACnetRM_BV := (Client:=Client,nObjectInstance:=34576);
	
	
	
	
	
	
	
	
	
	
	
	
	StartStopCommand_136: FB_BACnetRM_BO := (Client:=Client,nObjectInstance:=34817);
	StartStopStatus_136: FB_BACnetRM_BI := (Client:=Client,nObjectInstance:=34818);
	Alarm_136: FB_BACnetRM_BI := (Client:=Client,nObjectInstance:=34819);
	MalfunctionCode_136: FB_BACnetRM_MI := (Client:=Client,nObjectInstance:=34820);
	
	
	
	
	RoomTemp_136: FB_BACnetRM_AI := (Client:=Client,nObjectInstance:=34825);
	TempAdjust_136: FB_BACnetRM_AV := (Client:=Client,nObjectInstance:=34826);
	FilterSign_136: FB_BACnetRM_BI := (Client:=Client,nObjectInstance:=34827);
	FilterSignReset_136: FB_BACnetRM_BV := (Client:=Client,nObjectInstance:=34828);
	RemoteControlStart_136: FB_BACnetRM_BV := (Client:=Client,nObjectInstance:=34829);
	
	RemoteControlTempAdjust_136: FB_BACnetRM_BV := (Client:=Client,nObjectInstance:=34832);
	
	
	
	
	
	
	
	
	
	
	
	
	StartStopCommand_137: FB_BACnetRM_BO := (Client:=Client,nObjectInstance:=35073);
	StartStopStatus_137: FB_BACnetRM_BI := (Client:=Client,nObjectInstance:=35074);
	Alarm_137: FB_BACnetRM_BI := (Client:=Client,nObjectInstance:=35075);
	MalfunctionCode_137: FB_BACnetRM_MI := (Client:=Client,nObjectInstance:=35076);
	
	
	
	
	RoomTemp_137: FB_BACnetRM_AI := (Client:=Client,nObjectInstance:=35081);
	TempAdjust_137: FB_BACnetRM_AV := (Client:=Client,nObjectInstance:=35082);
	FilterSign_137: FB_BACnetRM_BI := (Client:=Client,nObjectInstance:=35083);
	FilterSignReset_137: FB_BACnetRM_BV := (Client:=Client,nObjectInstance:=35084);
	RemoteControlStart_137: FB_BACnetRM_BV := (Client:=Client,nObjectInstance:=35085);
	
	RemoteControlTempAdjust_137: FB_BACnetRM_BV := (Client:=Client,nObjectInstance:=35088);
	
	
	
	
	
	
	
	
	
	
	
	
	StartStopCommand_138: FB_BACnetRM_BO := (Client:=Client,nObjectInstance:=35329);
	StartStopStatus_138: FB_BACnetRM_BI := (Client:=Client,nObjectInstance:=35330);
	Alarm_138: FB_BACnetRM_BI := (Client:=Client,nObjectInstance:=35331);
	MalfunctionCode_138: FB_BACnetRM_MI := (Client:=Client,nObjectInstance:=35332);
	
	
	
	
	RoomTemp_138: FB_BACnetRM_AI := (Client:=Client,nObjectInstance:=35337);
	TempAdjust_138: FB_BACnetRM_AV := (Client:=Client,nObjectInstance:=35338);
	FilterSign_138: FB_BACnetRM_BI := (Client:=Client,nObjectInstance:=35339);
	FilterSignReset_138: FB_BACnetRM_BV := (Client:=Client,nObjectInstance:=35340);
	RemoteControlStart_138: FB_BACnetRM_BV := (Client:=Client,nObjectInstance:=35341);
	
	RemoteControlTempAdjust_138: FB_BACnetRM_BV := (Client:=Client,nObjectInstance:=35344);
	
	
	
	
	
	
	
	
	
	
	
	
	StartStopCommand_139: FB_BACnetRM_BO := (Client:=Client,nObjectInstance:=35585);
	StartStopStatus_139: FB_BACnetRM_BI := (Client:=Client,nObjectInstance:=35586);
	Alarm_139: FB_BACnetRM_BI := (Client:=Client,nObjectInstance:=35587);
	MalfunctionCode_139: FB_BACnetRM_MI := (Client:=Client,nObjectInstance:=35588);
	
	
	
	
	RoomTemp_139: FB_BACnetRM_AI := (Client:=Client,nObjectInstance:=35593);
	TempAdjust_139: FB_BACnetRM_AV := (Client:=Client,nObjectInstance:=35594);
	FilterSign_139: FB_BACnetRM_BI := (Client:=Client,nObjectInstance:=35595);
	FilterSignReset_139: FB_BACnetRM_BV := (Client:=Client,nObjectInstance:=35596);
	RemoteControlStart_139: FB_BACnetRM_BV := (Client:=Client,nObjectInstance:=35597);
	
	RemoteControlTempAdjust_139: FB_BACnetRM_BV := (Client:=Client,nObjectInstance:=35600);
	
	
	
	
	
	
	
	
	
	
	
	
	StartStopCommand_141: FB_BACnetRM_BO := (Client:=Client,nObjectInstance:=36097);
	StartStopStatus_141: FB_BACnetRM_BI := (Client:=Client,nObjectInstance:=36098);
	Alarm_141: FB_BACnetRM_BI := (Client:=Client,nObjectInstance:=36099);
	MalfunctionCode_141: FB_BACnetRM_MI := (Client:=Client,nObjectInstance:=36100);
	
	
	
	
	RoomTemp_141: FB_BACnetRM_AI := (Client:=Client,nObjectInstance:=36105);
	TempAdjust_141: FB_BACnetRM_AV := (Client:=Client,nObjectInstance:=36106);
	FilterSign_141: FB_BACnetRM_BI := (Client:=Client,nObjectInstance:=36107);
	FilterSignReset_141: FB_BACnetRM_BV := (Client:=Client,nObjectInstance:=36108);
	RemoteControlStart_141: FB_BACnetRM_BV := (Client:=Client,nObjectInstance:=36109);
	
	RemoteControlTempAdjust_141: FB_BACnetRM_BV := (Client:=Client,nObjectInstance:=36112);
	
	
	
	
	
	
	
	
	
	
	
	
	StartStopCommand_142: FB_BACnetRM_BO := (Client:=Client,nObjectInstance:=36353);
	StartStopStatus_142: FB_BACnetRM_BI := (Client:=Client,nObjectInstance:=36354);
	Alarm_142: FB_BACnetRM_BI := (Client:=Client,nObjectInstance:=36355);
	MalfunctionCode_142: FB_BACnetRM_MI := (Client:=Client,nObjectInstance:=36356);
	
	
	
	
	RoomTemp_142: FB_BACnetRM_AI := (Client:=Client,nObjectInstance:=36361);
	TempAdjust_142: FB_BACnetRM_AV := (Client:=Client,nObjectInstance:=36362);
	FilterSign_142: FB_BACnetRM_BI := (Client:=Client,nObjectInstance:=36363);
	FilterSignReset_142: FB_BACnetRM_BV := (Client:=Client,nObjectInstance:=36364);
	RemoteControlStart_142: FB_BACnetRM_BV := (Client:=Client,nObjectInstance:=36365);
	
	RemoteControlTempAdjust_142: FB_BACnetRM_BV := (Client:=Client,nObjectInstance:=36368);
	
	
	
	
	
	
	
	
	
	
	
	
	StartStopCommand_143: FB_BACnetRM_BO := (Client:=Client,nObjectInstance:=36609);
	StartStopStatus_143: FB_BACnetRM_BI := (Client:=Client,nObjectInstance:=36610);
	Alarm_143: FB_BACnetRM_BI := (Client:=Client,nObjectInstance:=36611);
	MalfunctionCode_143: FB_BACnetRM_MI := (Client:=Client,nObjectInstance:=36612);
	
	
	
	
	RoomTemp_143: FB_BACnetRM_AI := (Client:=Client,nObjectInstance:=36617);
	TempAdjust_143: FB_BACnetRM_AV := (Client:=Client,nObjectInstance:=36618);
	FilterSign_143: FB_BACnetRM_BI := (Client:=Client,nObjectInstance:=36619);
	FilterSignReset_143: FB_BACnetRM_BV := (Client:=Client,nObjectInstance:=36620);
	RemoteControlStart_143: FB_BACnetRM_BV := (Client:=Client,nObjectInstance:=36621);
	
	RemoteControlTempAdjust_143: FB_BACnetRM_BV := (Client:=Client,nObjectInstance:=36624);
	
	
	
	
	
	
	
	
	
	
	
	
	StartStopCommand_144: FB_BACnetRM_BO := (Client:=Client,nObjectInstance:=36865);
	StartStopStatus_144: FB_BACnetRM_BI := (Client:=Client,nObjectInstance:=36866);
	Alarm_144: FB_BACnetRM_BI := (Client:=Client,nObjectInstance:=36867);
	MalfunctionCode_144: FB_BACnetRM_MI := (Client:=Client,nObjectInstance:=36868);
	
	
	
	
	RoomTemp_144: FB_BACnetRM_AI := (Client:=Client,nObjectInstance:=36873);
	TempAdjust_144: FB_BACnetRM_AV := (Client:=Client,nObjectInstance:=36874);
	FilterSign_144: FB_BACnetRM_BI := (Client:=Client,nObjectInstance:=36875);
	FilterSignReset_144: FB_BACnetRM_BV := (Client:=Client,nObjectInstance:=36876);
	RemoteControlStart_144: FB_BACnetRM_BV := (Client:=Client,nObjectInstance:=36877);
	
	RemoteControlTempAdjust_144: FB_BACnetRM_BV := (Client:=Client,nObjectInstance:=36880);
	
	
	
	
	
	
	
	
	
	
	
	
	StartStopCommand_145: FB_BACnetRM_BO := (Client:=Client,nObjectInstance:=37121);
	StartStopStatus_145: FB_BACnetRM_BI := (Client:=Client,nObjectInstance:=37122);
	Alarm_145: FB_BACnetRM_BI := (Client:=Client,nObjectInstance:=37123);
	MalfunctionCode_145: FB_BACnetRM_MI := (Client:=Client,nObjectInstance:=37124);
	
	
	
	
	RoomTemp_145: FB_BACnetRM_AI := (Client:=Client,nObjectInstance:=37129);
	TempAdjust_145: FB_BACnetRM_AV := (Client:=Client,nObjectInstance:=37130);
	FilterSign_145: FB_BACnetRM_BI := (Client:=Client,nObjectInstance:=37131);
	FilterSignReset_145: FB_BACnetRM_BV := (Client:=Client,nObjectInstance:=37132);
	RemoteControlStart_145: FB_BACnetRM_BV := (Client:=Client,nObjectInstance:=37133);
	
	RemoteControlTempAdjust_145: FB_BACnetRM_BV := (Client:=Client,nObjectInstance:=37136);
	
	
	
	
	
	
	
	
	
	
	
	
	StartStopCommand_146: FB_BACnetRM_BO := (Client:=Client,nObjectInstance:=37377);
	StartStopStatus_146: FB_BACnetRM_BI := (Client:=Client,nObjectInstance:=37378);
	Alarm_146: FB_BACnetRM_BI := (Client:=Client,nObjectInstance:=37379);
	MalfunctionCode_146: FB_BACnetRM_MI := (Client:=Client,nObjectInstance:=37380);
	
	
	
	
	RoomTemp_146: FB_BACnetRM_AI := (Client:=Client,nObjectInstance:=37385);
	TempAdjust_146: FB_BACnetRM_AV := (Client:=Client,nObjectInstance:=37386);
	FilterSign_146: FB_BACnetRM_BI := (Client:=Client,nObjectInstance:=37387);
	FilterSignReset_146: FB_BACnetRM_BV := (Client:=Client,nObjectInstance:=37388);
	RemoteControlStart_146: FB_BACnetRM_BV := (Client:=Client,nObjectInstance:=37389);
	
	RemoteControlTempAdjust_146: FB_BACnetRM_BV := (Client:=Client,nObjectInstance:=37392);
	
	
	
	
	
	
	
	
	
	
	
	
	StartStopCommand_147: FB_BACnetRM_BO := (Client:=Client,nObjectInstance:=37633);
	StartStopStatus_147: FB_BACnetRM_BI := (Client:=Client,nObjectInstance:=37634);
	Alarm_147: FB_BACnetRM_BI := (Client:=Client,nObjectInstance:=37635);
	MalfunctionCode_147: FB_BACnetRM_MI := (Client:=Client,nObjectInstance:=37636);
	
	
	
	
	RoomTemp_147: FB_BACnetRM_AI := (Client:=Client,nObjectInstance:=37641);
	TempAdjust_147: FB_BACnetRM_AV := (Client:=Client,nObjectInstance:=37642);
	FilterSign_147: FB_BACnetRM_BI := (Client:=Client,nObjectInstance:=37643);
	FilterSignReset_147: FB_BACnetRM_BV := (Client:=Client,nObjectInstance:=37644);
	RemoteControlStart_147: FB_BACnetRM_BV := (Client:=Client,nObjectInstance:=37645);
	
	RemoteControlTempAdjust_147: FB_BACnetRM_BV := (Client:=Client,nObjectInstance:=37648);
	
	
	
	
	
	
	
	
	
	
	
	
	StartStopCommand_148: FB_BACnetRM_BO := (Client:=Client,nObjectInstance:=37889);
	StartStopStatus_148: FB_BACnetRM_BI := (Client:=Client,nObjectInstance:=37890);
	Alarm_148: FB_BACnetRM_BI := (Client:=Client,nObjectInstance:=37891);
	MalfunctionCode_148: FB_BACnetRM_MI := (Client:=Client,nObjectInstance:=37892);
	
	
	
	
	RoomTemp_148: FB_BACnetRM_AI := (Client:=Client,nObjectInstance:=37897);
	TempAdjust_148: FB_BACnetRM_AV := (Client:=Client,nObjectInstance:=37898);
	FilterSign_148: FB_BACnetRM_BI := (Client:=Client,nObjectInstance:=37899);
	FilterSignReset_148: FB_BACnetRM_BV := (Client:=Client,nObjectInstance:=37900);
	RemoteControlStart_148: FB_BACnetRM_BV := (Client:=Client,nObjectInstance:=37901);
	
	RemoteControlTempAdjust_148: FB_BACnetRM_BV := (Client:=Client,nObjectInstance:=37904);
	
	
	
	
	
	
	
	
	
	
	
	
	StartStopCommand_160: FB_BACnetRM_BO := (Client:=Client,nObjectInstance:=40961);
	StartStopStatus_160: FB_BACnetRM_BI := (Client:=Client,nObjectInstance:=40962);
	Alarm_160: FB_BACnetRM_BI := (Client:=Client,nObjectInstance:=40963);
	MalfunctionCode_160: FB_BACnetRM_MI := (Client:=Client,nObjectInstance:=40964);
	
	
	
	
	RoomTemp_160: FB_BACnetRM_AI := (Client:=Client,nObjectInstance:=40969);
	TempAdjust_160: FB_BACnetRM_AV := (Client:=Client,nObjectInstance:=40970);
	FilterSign_160: FB_BACnetRM_BI := (Client:=Client,nObjectInstance:=40971);
	FilterSignReset_160: FB_BACnetRM_BV := (Client:=Client,nObjectInstance:=40972);
	RemoteControlStart_160: FB_BACnetRM_BV := (Client:=Client,nObjectInstance:=40973);
	
	RemoteControlTempAdjust_160: FB_BACnetRM_BV := (Client:=Client,nObjectInstance:=40976);
	
	
	
	
	
	
	
	
	
	
	
	
	StartStopCommand_161: FB_BACnetRM_BO := (Client:=Client,nObjectInstance:=41217);
	StartStopStatus_161: FB_BACnetRM_BI := (Client:=Client,nObjectInstance:=41218);
	Alarm_161: FB_BACnetRM_BI := (Client:=Client,nObjectInstance:=41219);
	MalfunctionCode_161: FB_BACnetRM_MI := (Client:=Client,nObjectInstance:=41220);
	
	
	
	
	RoomTemp_161: FB_BACnetRM_AI := (Client:=Client,nObjectInstance:=41225);
	TempAdjust_161: FB_BACnetRM_AV := (Client:=Client,nObjectInstance:=41226);
	FilterSign_161: FB_BACnetRM_BI := (Client:=Client,nObjectInstance:=41227);
	FilterSignReset_161: FB_BACnetRM_BV := (Client:=Client,nObjectInstance:=41228);
	RemoteControlStart_161: FB_BACnetRM_BV := (Client:=Client,nObjectInstance:=41229);
	
	RemoteControlTempAdjust_161: FB_BACnetRM_BV := (Client:=Client,nObjectInstance:=41232);
	
	
	
	
	
	
	
	
	
	
	
	
	StartStopCommand_162: FB_BACnetRM_BO := (Client:=Client,nObjectInstance:=41473);
	StartStopStatus_162: FB_BACnetRM_BI := (Client:=Client,nObjectInstance:=41474);
	Alarm_162: FB_BACnetRM_BI := (Client:=Client,nObjectInstance:=41475);
	MalfunctionCode_162: FB_BACnetRM_MI := (Client:=Client,nObjectInstance:=41476);
	
	
	
	
	RoomTemp_162: FB_BACnetRM_AI := (Client:=Client,nObjectInstance:=41481);
	TempAdjust_162: FB_BACnetRM_AV := (Client:=Client,nObjectInstance:=41482);
	FilterSign_162: FB_BACnetRM_BI := (Client:=Client,nObjectInstance:=41483);
	FilterSignReset_162: FB_BACnetRM_BV := (Client:=Client,nObjectInstance:=41484);
	RemoteControlStart_162: FB_BACnetRM_BV := (Client:=Client,nObjectInstance:=41485);
	
	RemoteControlTempAdjust_162: FB_BACnetRM_BV := (Client:=Client,nObjectInstance:=41488);
	
	
	
	
	
	
	
	
	
	
	
	
	StartStopCommand_163: FB_BACnetRM_BO := (Client:=Client,nObjectInstance:=41729);
	StartStopStatus_163: FB_BACnetRM_BI := (Client:=Client,nObjectInstance:=41730);
	Alarm_163: FB_BACnetRM_BI := (Client:=Client,nObjectInstance:=41731);
	MalfunctionCode_163: FB_BACnetRM_MI := (Client:=Client,nObjectInstance:=41732);
	
	
	
	
	RoomTemp_163: FB_BACnetRM_AI := (Client:=Client,nObjectInstance:=41737);
	TempAdjust_163: FB_BACnetRM_AV := (Client:=Client,nObjectInstance:=41738);
	FilterSign_163: FB_BACnetRM_BI := (Client:=Client,nObjectInstance:=41739);
	FilterSignReset_163: FB_BACnetRM_BV := (Client:=Client,nObjectInstance:=41740);
	RemoteControlStart_163: FB_BACnetRM_BV := (Client:=Client,nObjectInstance:=41741);
	
	RemoteControlTempAdjust_163: FB_BACnetRM_BV := (Client:=Client,nObjectInstance:=41744);
	
	
	
	
	
	
	
	
	
	
	
	
	StartStopCommand_164: FB_BACnetRM_BO := (Client:=Client,nObjectInstance:=41985);
	StartStopStatus_164: FB_BACnetRM_BI := (Client:=Client,nObjectInstance:=41986);
	Alarm_164: FB_BACnetRM_BI := (Client:=Client,nObjectInstance:=41987);
	MalfunctionCode_164: FB_BACnetRM_MI := (Client:=Client,nObjectInstance:=41988);
	
	
	
	
	RoomTemp_164: FB_BACnetRM_AI := (Client:=Client,nObjectInstance:=41993);
	TempAdjust_164: FB_BACnetRM_AV := (Client:=Client,nObjectInstance:=41994);
	FilterSign_164: FB_BACnetRM_BI := (Client:=Client,nObjectInstance:=41995);
	FilterSignReset_164: FB_BACnetRM_BV := (Client:=Client,nObjectInstance:=41996);
	RemoteControlStart_164: FB_BACnetRM_BV := (Client:=Client,nObjectInstance:=41997);
	
	RemoteControlTempAdjust_164: FB_BACnetRM_BV := (Client:=Client,nObjectInstance:=42000);
	
	
	
	
	
	
	
	
	
	
	
	
	StartStopCommand_165: FB_BACnetRM_BO := (Client:=Client,nObjectInstance:=42241);
	StartStopStatus_165: FB_BACnetRM_BI := (Client:=Client,nObjectInstance:=42242);
	Alarm_165: FB_BACnetRM_BI := (Client:=Client,nObjectInstance:=42243);
	MalfunctionCode_165: FB_BACnetRM_MI := (Client:=Client,nObjectInstance:=42244);
	
	
	
	
	RoomTemp_165: FB_BACnetRM_AI := (Client:=Client,nObjectInstance:=42249);
	TempAdjust_165: FB_BACnetRM_AV := (Client:=Client,nObjectInstance:=42250);
	FilterSign_165: FB_BACnetRM_BI := (Client:=Client,nObjectInstance:=42251);
	FilterSignReset_165: FB_BACnetRM_BV := (Client:=Client,nObjectInstance:=42252);
	RemoteControlStart_165: FB_BACnetRM_BV := (Client:=Client,nObjectInstance:=42253);
	
	RemoteControlTempAdjust_165: FB_BACnetRM_BV := (Client:=Client,nObjectInstance:=42256);
	
	
	
	
	
	
	
	
	
	
	
	
	StartStopCommand_166: FB_BACnetRM_BO := (Client:=Client,nObjectInstance:=42497);
	StartStopStatus_166: FB_BACnetRM_BI := (Client:=Client,nObjectInstance:=42498);
	Alarm_166: FB_BACnetRM_BI := (Client:=Client,nObjectInstance:=42499);
	MalfunctionCode_166: FB_BACnetRM_MI := (Client:=Client,nObjectInstance:=42500);
	
	
	
	
	RoomTemp_166: FB_BACnetRM_AI := (Client:=Client,nObjectInstance:=42505);
	TempAdjust_166: FB_BACnetRM_AV := (Client:=Client,nObjectInstance:=42506);
	FilterSign_166: FB_BACnetRM_BI := (Client:=Client,nObjectInstance:=42507);
	FilterSignReset_166: FB_BACnetRM_BV := (Client:=Client,nObjectInstance:=42508);
	RemoteControlStart_166: FB_BACnetRM_BV := (Client:=Client,nObjectInstance:=42509);
	
	RemoteControlTempAdjust_166: FB_BACnetRM_BV := (Client:=Client,nObjectInstance:=42512);
	
	
	
	
	
	
	
	
	
	
	
	
	StartStopCommand_167: FB_BACnetRM_BO := (Client:=Client,nObjectInstance:=42753);
	StartStopStatus_167: FB_BACnetRM_BI := (Client:=Client,nObjectInstance:=42754);
	Alarm_167: FB_BACnetRM_BI := (Client:=Client,nObjectInstance:=42755);
	MalfunctionCode_167: FB_BACnetRM_MI := (Client:=Client,nObjectInstance:=42756);
	
	
	
	
	RoomTemp_167: FB_BACnetRM_AI := (Client:=Client,nObjectInstance:=42761);
	TempAdjust_167: FB_BACnetRM_AV := (Client:=Client,nObjectInstance:=42762);
	FilterSign_167: FB_BACnetRM_BI := (Client:=Client,nObjectInstance:=42763);
	FilterSignReset_167: FB_BACnetRM_BV := (Client:=Client,nObjectInstance:=42764);
	RemoteControlStart_167: FB_BACnetRM_BV := (Client:=Client,nObjectInstance:=42765);
	
	RemoteControlTempAdjust_167: FB_BACnetRM_BV := (Client:=Client,nObjectInstance:=42768);
	
	
	
	
	
	
	
	
	
	
	
	
	StartStopCommand_176: FB_BACnetRM_BO := (Client:=Client,nObjectInstance:=45057);
	StartStopStatus_176: FB_BACnetRM_BI := (Client:=Client,nObjectInstance:=45058);
	Alarm_176: FB_BACnetRM_BI := (Client:=Client,nObjectInstance:=45059);
	MalfunctionCode_176: FB_BACnetRM_MI := (Client:=Client,nObjectInstance:=45060);
	
	
	
	
	RoomTemp_176: FB_BACnetRM_AI := (Client:=Client,nObjectInstance:=45065);
	TempAdjust_176: FB_BACnetRM_AV := (Client:=Client,nObjectInstance:=45066);
	FilterSign_176: FB_BACnetRM_BI := (Client:=Client,nObjectInstance:=45067);
	FilterSignReset_176: FB_BACnetRM_BV := (Client:=Client,nObjectInstance:=45068);
	RemoteControlStart_176: FB_BACnetRM_BV := (Client:=Client,nObjectInstance:=45069);
	
	RemoteControlTempAdjust_176: FB_BACnetRM_BV := (Client:=Client,nObjectInstance:=45072);
	
	
	
	
	
	
	
	
	
	
	
	
	StartStopCommand_193: FB_BACnetRM_BO := (Client:=Client,nObjectInstance:=49409);
	StartStopStatus_193: FB_BACnetRM_BI := (Client:=Client,nObjectInstance:=49410);
	Alarm_193: FB_BACnetRM_BI := (Client:=Client,nObjectInstance:=49411);
	MalfunctionCode_193: FB_BACnetRM_MI := (Client:=Client,nObjectInstance:=49412);
	
	
	
	
	RoomTemp_193: FB_BACnetRM_AI := (Client:=Client,nObjectInstance:=49417);
	TempAdjust_193: FB_BACnetRM_AV := (Client:=Client,nObjectInstance:=49418);
	FilterSign_193: FB_BACnetRM_BI := (Client:=Client,nObjectInstance:=49419);
	FilterSignReset_193: FB_BACnetRM_BV := (Client:=Client,nObjectInstance:=49420);
	RemoteControlStart_193: FB_BACnetRM_BV := (Client:=Client,nObjectInstance:=49421);
	
	RemoteControlTempAdjust_193: FB_BACnetRM_BV := (Client:=Client,nObjectInstance:=49424);
	
	
	
	
	
	
	
	
	
	
	
	
	StartStopCommand_194: FB_BACnetRM_BO := (Client:=Client,nObjectInstance:=49665);
	StartStopStatus_194: FB_BACnetRM_BI := (Client:=Client,nObjectInstance:=49666);
	Alarm_194: FB_BACnetRM_BI := (Client:=Client,nObjectInstance:=49667);
	MalfunctionCode_194: FB_BACnetRM_MI := (Client:=Client,nObjectInstance:=49668);
	
	
	
	
	RoomTemp_194: FB_BACnetRM_AI := (Client:=Client,nObjectInstance:=49673);
	TempAdjust_194: FB_BACnetRM_AV := (Client:=Client,nObjectInstance:=49674);
	FilterSign_194: FB_BACnetRM_BI := (Client:=Client,nObjectInstance:=49675);
	FilterSignReset_194: FB_BACnetRM_BV := (Client:=Client,nObjectInstance:=49676);
	RemoteControlStart_194: FB_BACnetRM_BV := (Client:=Client,nObjectInstance:=49677);
	
	RemoteControlTempAdjust_194: FB_BACnetRM_BV := (Client:=Client,nObjectInstance:=49680);
	
	
	
	
	
	
	
	
	
	
	
	
	StartStopCommand_195: FB_BACnetRM_BO := (Client:=Client,nObjectInstance:=49921);
	StartStopStatus_195: FB_BACnetRM_BI := (Client:=Client,nObjectInstance:=49922);
	Alarm_195: FB_BACnetRM_BI := (Client:=Client,nObjectInstance:=49923);
	MalfunctionCode_195: FB_BACnetRM_MI := (Client:=Client,nObjectInstance:=49924);
	
	
	
	
	RoomTemp_195: FB_BACnetRM_AI := (Client:=Client,nObjectInstance:=49929);
	TempAdjust_195: FB_BACnetRM_AV := (Client:=Client,nObjectInstance:=49930);
	FilterSign_195: FB_BACnetRM_BI := (Client:=Client,nObjectInstance:=49931);
	FilterSignReset_195: FB_BACnetRM_BV := (Client:=Client,nObjectInstance:=49932);
	RemoteControlStart_195: FB_BACnetRM_BV := (Client:=Client,nObjectInstance:=49933);
	
	RemoteControlTempAdjust_195: FB_BACnetRM_BV := (Client:=Client,nObjectInstance:=49936);
	
	
	
	
	
	
	
	
	
	
	
	
	StartStopCommand_196: FB_BACnetRM_BO := (Client:=Client,nObjectInstance:=50177);
	StartStopStatus_196: FB_BACnetRM_BI := (Client:=Client,nObjectInstance:=50178);
	Alarm_196: FB_BACnetRM_BI := (Client:=Client,nObjectInstance:=50179);
	MalfunctionCode_196: FB_BACnetRM_MI := (Client:=Client,nObjectInstance:=50180);
	
	
	
	
	RoomTemp_196: FB_BACnetRM_AI := (Client:=Client,nObjectInstance:=50185);
	TempAdjust_196: FB_BACnetRM_AV := (Client:=Client,nObjectInstance:=50186);
	FilterSign_196: FB_BACnetRM_BI := (Client:=Client,nObjectInstance:=50187);
	FilterSignReset_196: FB_BACnetRM_BV := (Client:=Client,nObjectInstance:=50188);
	RemoteControlStart_196: FB_BACnetRM_BV := (Client:=Client,nObjectInstance:=50189);
	
	RemoteControlTempAdjust_196: FB_BACnetRM_BV := (Client:=Client,nObjectInstance:=50192);
	
	
	
	
	
	
	
	
	
	
	
	
	StartStopCommand_197: FB_BACnetRM_BO := (Client:=Client,nObjectInstance:=50433);
	StartStopStatus_197: FB_BACnetRM_BI := (Client:=Client,nObjectInstance:=50434);
	Alarm_197: FB_BACnetRM_BI := (Client:=Client,nObjectInstance:=50435);
	MalfunctionCode_197: FB_BACnetRM_MI := (Client:=Client,nObjectInstance:=50436);
	
	
	
	
	RoomTemp_197: FB_BACnetRM_AI := (Client:=Client,nObjectInstance:=50441);
	TempAdjust_197: FB_BACnetRM_AV := (Client:=Client,nObjectInstance:=50442);
	FilterSign_197: FB_BACnetRM_BI := (Client:=Client,nObjectInstance:=50443);
	FilterSignReset_197: FB_BACnetRM_BV := (Client:=Client,nObjectInstance:=50444);
	RemoteControlStart_197: FB_BACnetRM_BV := (Client:=Client,nObjectInstance:=50445);
	
	RemoteControlTempAdjust_197: FB_BACnetRM_BV := (Client:=Client,nObjectInstance:=50448);
	
	
	
	
	
	
	
	
	
	
	
	
	StartStopCommand_198: FB_BACnetRM_BO := (Client:=Client,nObjectInstance:=50689);
	StartStopStatus_198: FB_BACnetRM_BI := (Client:=Client,nObjectInstance:=50690);
	Alarm_198: FB_BACnetRM_BI := (Client:=Client,nObjectInstance:=50691);
	MalfunctionCode_198: FB_BACnetRM_MI := (Client:=Client,nObjectInstance:=50692);
	
	
	
	
	RoomTemp_198: FB_BACnetRM_AI := (Client:=Client,nObjectInstance:=50697);
	TempAdjust_198: FB_BACnetRM_AV := (Client:=Client,nObjectInstance:=50698);
	FilterSign_198: FB_BACnetRM_BI := (Client:=Client,nObjectInstance:=50699);
	FilterSignReset_198: FB_BACnetRM_BV := (Client:=Client,nObjectInstance:=50700);
	RemoteControlStart_198: FB_BACnetRM_BV := (Client:=Client,nObjectInstance:=50701);
	
	RemoteControlTempAdjust_198: FB_BACnetRM_BV := (Client:=Client,nObjectInstance:=50704);
	
	
	
	
	
	
	
	
	
	
	
	
	StartStopCommand_199: FB_BACnetRM_BO := (Client:=Client,nObjectInstance:=50945);
	StartStopStatus_199: FB_BACnetRM_BI := (Client:=Client,nObjectInstance:=50946);
	Alarm_199: FB_BACnetRM_BI := (Client:=Client,nObjectInstance:=50947);
	MalfunctionCode_199: FB_BACnetRM_MI := (Client:=Client,nObjectInstance:=50948);
	
	
	
	
	RoomTemp_199: FB_BACnetRM_AI := (Client:=Client,nObjectInstance:=50953);
	TempAdjust_199: FB_BACnetRM_AV := (Client:=Client,nObjectInstance:=50954);
	FilterSign_199: FB_BACnetRM_BI := (Client:=Client,nObjectInstance:=50955);
	FilterSignReset_199: FB_BACnetRM_BV := (Client:=Client,nObjectInstance:=50956);
	RemoteControlStart_199: FB_BACnetRM_BV := (Client:=Client,nObjectInstance:=50957);
	
	RemoteControlTempAdjust_199: FB_BACnetRM_BV := (Client:=Client,nObjectInstance:=50960);
	
	
	
	
	
	
	
	
	
	
	
	
	StartStopCommand_200: FB_BACnetRM_BO := (Client:=Client,nObjectInstance:=51201);
	StartStopStatus_200: FB_BACnetRM_BI := (Client:=Client,nObjectInstance:=51202);
	Alarm_200: FB_BACnetRM_BI := (Client:=Client,nObjectInstance:=51203);
	MalfunctionCode_200: FB_BACnetRM_MI := (Client:=Client,nObjectInstance:=51204);
	
	
	
	
	RoomTemp_200: FB_BACnetRM_AI := (Client:=Client,nObjectInstance:=51209);
	TempAdjust_200: FB_BACnetRM_AV := (Client:=Client,nObjectInstance:=51210);
	FilterSign_200: FB_BACnetRM_BI := (Client:=Client,nObjectInstance:=51211);
	FilterSignReset_200: FB_BACnetRM_BV := (Client:=Client,nObjectInstance:=51212);
	RemoteControlStart_200: FB_BACnetRM_BV := (Client:=Client,nObjectInstance:=51213);
	
	RemoteControlTempAdjust_200: FB_BACnetRM_BV := (Client:=Client,nObjectInstance:=51216);
	
	
	
	
	
	
	
	
	
	
	
	
	StartStopCommand_201: FB_BACnetRM_BO := (Client:=Client,nObjectInstance:=51457);
	StartStopStatus_201: FB_BACnetRM_BI := (Client:=Client,nObjectInstance:=51458);
	Alarm_201: FB_BACnetRM_BI := (Client:=Client,nObjectInstance:=51459);
	MalfunctionCode_201: FB_BACnetRM_MI := (Client:=Client,nObjectInstance:=51460);
	
	
	
	
	RoomTemp_201: FB_BACnetRM_AI := (Client:=Client,nObjectInstance:=51465);
	TempAdjust_201: FB_BACnetRM_AV := (Client:=Client,nObjectInstance:=51466);
	FilterSign_201: FB_BACnetRM_BI := (Client:=Client,nObjectInstance:=51467);
	FilterSignReset_201: FB_BACnetRM_BV := (Client:=Client,nObjectInstance:=51468);
	RemoteControlStart_201: FB_BACnetRM_BV := (Client:=Client,nObjectInstance:=51469);
	
	RemoteControlTempAdjust_201: FB_BACnetRM_BV := (Client:=Client,nObjectInstance:=51472);
	
	
	
	
	
	
	
	
	
	
	
	
	StartStopCommand_202: FB_BACnetRM_BO := (Client:=Client,nObjectInstance:=51713);
	StartStopStatus_202: FB_BACnetRM_BI := (Client:=Client,nObjectInstance:=51714);
	Alarm_202: FB_BACnetRM_BI := (Client:=Client,nObjectInstance:=51715);
	MalfunctionCode_202: FB_BACnetRM_MI := (Client:=Client,nObjectInstance:=51716);
	
	
	
	
	RoomTemp_202: FB_BACnetRM_AI := (Client:=Client,nObjectInstance:=51721);
	TempAdjust_202: FB_BACnetRM_AV := (Client:=Client,nObjectInstance:=51722);
	FilterSign_202: FB_BACnetRM_BI := (Client:=Client,nObjectInstance:=51723);
	FilterSignReset_202: FB_BACnetRM_BV := (Client:=Client,nObjectInstance:=51724);
	RemoteControlStart_202: FB_BACnetRM_BV := (Client:=Client,nObjectInstance:=51725);
	
	RemoteControlTempAdjust_202: FB_BACnetRM_BV := (Client:=Client,nObjectInstance:=51728);
	
	
	
	
	
	
	
	
	
	
	
	
	StartStopCommand_203: FB_BACnetRM_BO := (Client:=Client,nObjectInstance:=51969);
	StartStopStatus_203: FB_BACnetRM_BI := (Client:=Client,nObjectInstance:=51970);
	Alarm_203: FB_BACnetRM_BI := (Client:=Client,nObjectInstance:=51971);
	MalfunctionCode_203: FB_BACnetRM_MI := (Client:=Client,nObjectInstance:=51972);
	
	
	
	
	RoomTemp_203: FB_BACnetRM_AI := (Client:=Client,nObjectInstance:=51977);
	TempAdjust_203: FB_BACnetRM_AV := (Client:=Client,nObjectInstance:=51978);
	FilterSign_203: FB_BACnetRM_BI := (Client:=Client,nObjectInstance:=51979);
	FilterSignReset_203: FB_BACnetRM_BV := (Client:=Client,nObjectInstance:=51980);
	RemoteControlStart_203: FB_BACnetRM_BV := (Client:=Client,nObjectInstance:=51981);
	
	RemoteControlTempAdjust_203: FB_BACnetRM_BV := (Client:=Client,nObjectInstance:=51984);
	
	
	
	
	
	
	
	
	
	
	
	
	StartStopCommand_204: FB_BACnetRM_BO := (Client:=Client,nObjectInstance:=52225);
	StartStopStatus_204: FB_BACnetRM_BI := (Client:=Client,nObjectInstance:=52226);
	Alarm_204: FB_BACnetRM_BI := (Client:=Client,nObjectInstance:=52227);
	MalfunctionCode_204: FB_BACnetRM_MI := (Client:=Client,nObjectInstance:=52228);
	
	
	
	
